LIN {X 0,Y 206.175,Z 893.981,A -85,B 0,C 180,E1 -23802.983,E2 -23802.983} C_VEL
LIN {X 0,Y 205.634,Z 894.543,A -85,B 0,C 180,E1 -23804.133,E2 -23804.133} C_VEL
LIN {X 0,Y 204.142,Z 895.622,A -85,B 0,C 180,E1 -23805.109,E2 -23805.109} C_VEL
LIN {X 0,Y 198.321,Z 899.43,A -85,B 0,C 180,E1 -23807.677,E2 -23807.677} C_VEL
LIN {X 0,Y 191.857,Z 903.186,A -85,B 0,C 180,E1 -23810.13,E2 -23810.13} C_VEL
LIN {X 0,Y 180.969,Z 908.434,A -85,B 0,C 180,E1 -23814.371,E2 -23814.371} C_VEL
LIN {X 0,Y 173.411,Z 911.413,A -85,B 0,C 180,E1 -23818.206,E2 -23818.206} C_VEL
LIN {X 0,Y 167.081,Z 913.319,A -85,B 0,C 180,E1 -23822.439,E2 -23822.439} C_VEL
LIN {X 0,Y 162.116,Z 914.142,A -85,B 0,C 180,E1 -23827.035,E2 -23827.035} C_VEL
LIN {X 0,Y 158.497,Z 913.842,A -85,B 0,C 180,E1 -23831.917,E2 -23831.917} C_VEL
LIN {X 0,Y 156.515,Z 912.431,A -85,B 0,C 180,E1 -23837.026,E2 -23837.026} C_VEL
LIN {X 0,Y 156.028,Z 909.791,A -85,B 0,C 180,E1 -23842.301,E2 -23842.301} C_VEL
LIN {X 0,Y 156.626,Z 905.821,A -85,B 0,C 180,E1 -23847.428,E2 -23847.428} C_VEL
LIN {X 0,Y 157.151,Z 904.017,A -85,B 0,C 180,E1 -23849.359,E2 -23849.359} C_VEL
LIN {X 0,Y 156.522,Z 907.281,A -85,B 0,C 180,E1 -23852.574,E2 -23852.574} C_VEL
LIN {X 0,Y 155.932,Z 911.226,A -85,B 0,C 180,E1 -23857.771,E2 -23857.771} C_VEL
LIN {X 0,Y 156.49,Z 913.74,A -85,B 0,C 180,E1 -23862.977,E2 -23862.977} C_VEL
LIN {X 0,Y 158.478,Z 915.084,A -85,B 0,C 180,E1 -23868.085,E2 -23868.085} C_VEL
LIN {X 0,Y 162.105,Z 915.337,A -85,B 0,C 180,E1 -23872.966,E2 -23872.966} C_VEL
LIN {X 0,Y 167.061,Z 914.483,A -85,B 0,C 180,E1 -23877.565,E2 -23877.565} C_VEL
LIN {X 0,Y 173.716,Z 912.427,A -85,B 0,C 180,E1 -23882.007,E2 -23882.007} C_VEL
LIN {X 0,Y 180.79,Z 909.587,A -85,B 0,C 180,E1 -23885.67,E2 -23885.67} C_VEL
LIN {X 0,Y 189.558,Z 905.487,A -85,B 0,C 180,E1 -23889.072,E2 -23889.072} C_VEL
LIN {X 0,Y 191.177,Z 904.654,A -85,B 0,C 180,E1 -23889.633,E2 -23889.633} C_VEL
LIN {X 0,Y 192.985,Z 903.559,A -85,B 0,C 180,E1 -23890.605,E2 -23890.605} C_VEL
LIN {X 0,Y 193.846,Z 902.733,A -85,B 0,C 180,E1 -23891.725,E2 -23891.725} C_VEL
LIN {X 0,Y 195.209,Z 900.797,A -85,B 0,C 180,E1 -23895.095,E2 -23895.095} C_VEL
LIN {X 0,Y 195.881,Z 900.333,A -85,B 0,C 180,E1 -23895.652,E2 -23895.652} C_VEL
LIN {X 0,Y 196.934,Z 899.471,A -85,B 0,C 180,E1 -23897.306,E2 -23897.306} C_VEL
LIN {X 0,Y 197.063,Z 899.174,A -85,B 0,C 180,E1 -23898.499,E2 -23898.499} C_VEL
LIN {X 0,Y 195.662,Z 899.564,A -85,B 0,C 180,E1 -23899.716,E2 -23899.716} C_VEL
LIN {X 0,Y 185.93,Z 902.848,A -85,B 0,C 180,E1 -23902.784,E2 -23902.784} C_VEL
LIN {X 0,Y 177.174,Z 904.928,A -85,B 0,C 180,E1 -23906.263,E2 -23906.263} C_VEL
LIN {X 0,Y 169.371,Z 905.875,A -85,B 0,C 180,E1 -23910.134,E2 -23910.134} C_VEL
LIN {X 0,Y 162.669,Z 905.677,A -85,B 0,C 180,E1 -23914.4,E2 -23914.4} C_VEL
LIN {X 0,Y 157.172,Z 904.299,A -85,B 0,C 180,E1 -23919.037,E2 -23919.037} C_VEL
LIN {X 0,Y 153.143,Z 901.751,A -85,B 0,C 180,E1 -23924.014,E2 -23924.014} C_VEL
LIN {X 0,Y 149.972,Z 897.499,A -85,B 0,C 180,E1 -23929.771,E2 -23929.771} C_VEL
LIN {X 0,Y 148.887,Z 892.858,A -85,B 0,C 180,E1 -23934.58,E2 -23934.58} C_VEL
LIN {X 0,Y 148.452,Z 887.997,A -85,B 0,C 180,E1 -23938.641,E2 -23938.641} C_VEL
LIN {X 0,Y 148.396,Z 882.089,A -85,B 0,C 180,E1 -23942.712,E2 -23942.712} C_VEL
LIN {X 0,Y 148.841,Z 873.681,A -85,B 0,C 180,E1 -23947.436,E2 -23947.436} C_VEL
LIN {X 0,Y 149.913,Z 863.17,A -85,B 0,C 180,E1 -23952.176,E2 -23952.176} C_VEL
LIN {X 0,Y 151.219,Z 853.005,A -85,B 0,C 180,E1 -23955.843,E2 -23955.843} C_VEL
LIN {X 0,Y 152.813,Z 841.876,A -85,B 0,C 180,E1 -23959.125,E2 -23959.125} C_VEL
LIN {X 0,Y 154.364,Z 831.542,A -85,B 0,C 180,E1 -23961.643,E2 -23961.643} C_VEL
LIN {X 0,Y 153.48,Z 825.601,A -85,B 0,C 180,E1 -23962.901,E2 -23962.901} C_VEL
LIN {X 0,Y 150.949,Z 811.534,A -85,B 0,C 180,E1 -23965.447,E2 -23965.447} C_VEL
LIN {X 0,Y 149.36,Z 802.881,A -85,B 0,C 180,E1 -23966.789,E2 -23966.789} C_VEL
LIN {X 0,Y 149.696,Z 802.832,A -85,B 0,C 180,E1 -23972.32,E2 -23972.32} C_VEL
LIN {X 0,Y 150.026,Z 802.795,A -85,B 0,C 180,E1 -23977.512,E2 -23977.512} C_VEL
LIN {X 0,Y 150.112,Z 802.781,A -85,B 0,C 180,E1 -23981.488,E2 -23981.488} C_VEL
LIN {X 0,Y 150.121,Z 802.784,A -85,B 0,C 180,E1 -23985.393,E2 -23985.393} C_VEL
LIN {X 0,Y 150.135,Z 802.777,A -85,B 0,C 180,E1 -23989.053,E2 -23989.053} C_VEL
LIN {X 0,Y 150.176,Z 802.777,A -85,B 0,C 180,E1 -23992.704,E2 -23992.704} C_VEL
LIN {X 0,Y 150.199,Z 802.77,A -85,B 0,C 180,E1 -23997.372,E2 -23997.372} C_VEL
LIN {X 0,Y 150.231,Z 802.771,A -85,B 0,C 180,E1 -24002.721,E2 -24002.721} C_VEL
LIN {X 0,Y 150.332,Z 802.755,A -85,B 0,C 180,E1 -24009.219,E2 -24009.219} C_VEL
LIN {X 0,Y 150.322,Z 802.759,A -85,B 0,C 180,E1 -24013.709,E2 -24013.709} C_VEL
LIN {X 0,Y 150.6,Z 802.723,A -85,B 0,C 180,E1 -24019.242,E2 -24019.242} C_VEL
LIN {X 0,Y 150.689,Z 802.714,A -85,B 0,C 180,E1 -24021.957,E2 -24021.957} C_VEL
LIN {X 0,Y 151.187,Z 802.654,A -85,B 0,C 180,E1 -24030,E2 -24030} C_VEL
LIN {X 0,Y 150.688,Z 802.714,A -85,B 0,C 180,E1 -24038.043,E2 -24038.043} C_VEL
LIN {X 0,Y 150.566,Z 802.727,A -85,B 0,C 180,E1 -24041.431,E2 -24041.431} C_VEL
LIN {X 0,Y 150.321,Z 802.759,A -85,B 0,C 180,E1 -24046.291,E2 -24046.291} C_VEL
LIN {X 0,Y 150.332,Z 802.755,A -85,B 0,C 180,E1 -24050.781,E2 -24050.781} C_VEL
LIN {X 0,Y 150.231,Z 802.771,A -85,B 0,C 180,E1 -24057.279,E2 -24057.279} C_VEL
LIN {X 0,Y 150.199,Z 802.77,A -85,B 0,C 180,E1 -24062.628,E2 -24062.628} C_VEL
LIN {X 0,Y 150.171,Z 802.777,A -85,B 0,C 180,E1 -24067.474,E2 -24067.474} C_VEL
LIN {X 0,Y 150.131,Z 802.78,A -85,B 0,C 180,E1 -24071.501,E2 -24071.501} C_VEL
LIN {X 0,Y 150.121,Z 802.786,A -85,B 0,C 180,E1 -24075.398,E2 -24075.398} C_VEL
LIN {X 0,Y 150.115,Z 802.781,A -85,B 0,C 180,E1 -24079.051,E2 -24079.051} C_VEL
LIN {X 0,Y 150.071,Z 802.79,A -85,B 0,C 180,E1 -24082.762,E2 -24082.762} C_VEL
LIN {X 0,Y 149.745,Z 802.826,A -85,B 0,C 180,E1 -24087.65,E2 -24087.65} C_VEL
LIN {X 0,Y 149.352,Z 802.883,A -85,B 0,C 180,E1 -24093.744,E2 -24093.744} C_VEL
LIN {X 0,Y 152.014,Z 817.45,A -85,B 0,C 180,E1 -24096.055,E2 -24096.055} C_VEL
LIN {X 0,Y 154.184,Z 829.238,A -85,B 0,C 180,E1 -24098.359,E2 -24098.359} C_VEL
LIN {X 0,Y 153.922,Z 833.391,A -85,B 0,C 180,E1 -24099.279,E2 -24099.279} C_VEL
LIN {X 0,Y 152.059,Z 845.938,A -85,B 0,C 180,E1 -24102.52,E2 -24102.52} C_VEL
LIN {X 0,Y 150.354,Z 858.144,A -85,B 0,C 180,E1 -24106.487,E2 -24106.487} C_VEL
LIN {X 0,Y 149.249,Z 868.043,A -85,B 0,C 180,E1 -24110.517,E2 -24110.517} C_VEL
LIN {X 0,Y 148.552,Z 876.986,A -85,B 0,C 180,E1 -24114.974,E2 -24114.974} C_VEL
LIN {X 0,Y 148.378,Z 883.073,A -85,B 0,C 180,E1 -24118.646,E2 -24118.646} C_VEL
LIN {X 0,Y 148.552,Z 888.659,A -85,B 0,C 180,E1 -24122.714,E2 -24122.714} C_VEL
LIN {X 0,Y 149.045,Z 893.275,A -85,B 0,C 180,E1 -24126.773,E2 -24126.773} C_VEL
LIN {X 0,Y 150.698,Z 898.09,A -85,B 0,C 180,E1 -24132.117,E2 -24132.117} C_VEL
LIN {X 0,Y 152.999,Z 900.836,A -85,B 0,C 180,E1 -24136.001,E2 -24136.001} C_VEL
LIN {X 0,Y 157.026,Z 903.417,A -85,B 0,C 180,E1 -24140.983,E2 -24140.983} C_VEL
LIN {X 0,Y 162.377,Z 904.818,A -85,B 0,C 180,E1 -24145.649,E2 -24145.649} C_VEL
LIN {X 0,Y 169.143,Z 905.029,A -85,B 0,C 180,E1 -24149.91,E2 -24149.91} C_VEL
LIN {X 0,Y 176.938,Z 904.069,A -85,B 0,C 180,E1 -24153.788,E2 -24153.788} C_VEL
LIN {X 0,Y 185.698,Z 901.963,A -85,B 0,C 180,E1 -24157.27,E2 -24157.27} C_VEL
LIN {X 0,Y 195.419,Z 898.667,A -85,B 0,C 180,E1 -24160.344,E2 -24160.344} C_VEL
LIN {X 0,Y 199.621,Z 897.048,A -85,B 0,C 180,E1 -24161.987,E2 -24161.987} C_VEL
LIN {X 0,Y 199.165,Z 897.595,A -85,B 0,C 180,E1 -24163.665,E2 -24163.665} C_VEL
LIN {X 0,Y 195.304,Z 899.854,A -85,B 0,C 180,E1 -24165.436,E2 -24165.436} C_VEL
LIN {X 0,Y 188.843,Z 903.25,A -85,B 0,C 180,E1 -24167.941,E2 -24167.941} C_VEL
LIN {X 0,Y 179.655,Z 907.311,A -85,B 0,C 180,E1 -24171.251,E2 -24171.251} C_VEL
LIN {X 0,Y 171.192,Z 910.365,A -85,B 0,C 180,E1 -24174.918,E2 -24174.918} C_VEL
LIN {X 0,Y 163.925,Z 912.373,A -85,B 0,C 180,E1 -24179.037,E2 -24179.037} C_VEL
LIN {X 0,Y 158.081,Z 913.344,A -85,B 0,C 180,E1 -24183.603,E2 -24183.603} C_VEL
LIN {X 0,Y 153.577,Z 913.247,A -85,B 0,C 180,E1 -24188.525,E2 -24188.525} C_VEL
LIN {X 0,Y 150.576,Z 912.07,A -85,B 0,C 180,E1 -24193.737,E2 -24193.737} C_VEL
LIN {X 0,Y 149.222,Z 909.786,A -85,B 0,C 180,E1 -24199.141,E2 -24199.141} C_VEL
LIN {X 0,Y 149.324,Z 906.261,A -85,B 0,C 180,E1 -24204.599,E2 -24204.599} C_VEL
LIN {X 0,Y 150.365,Z 901.963,A -85,B 0,C 180,E1 -24209.414,E2 -24209.414} C_VEL
LIN {X 0,Y 149.685,Z 905.392,A -85,B 0,C 180,E1 -24212.691,E2 -24212.691} C_VEL
LIN {X 0,Y 149.092,Z 909.56,A -85,B 0,C 180,E1 -24218.13,E2 -24218.13} C_VEL
LIN {X 0,Y 149.665,Z 912.382,A -85,B 0,C 180,E1 -24223.579,E2 -24223.579} C_VEL
LIN {X 0,Y 151.805,Z 914.025,A -85,B 0,C 180,E1 -24228.91,E2 -24228.91} C_VEL
LIN {X 0,Y 155.624,Z 914.615,A -85,B 0,C 180,E1 -24233.982,E2 -24233.982} C_VEL
LIN {X 0,Y 160.793,Z 914.136,A -85,B 0,C 180,E1 -24238.737,E2 -24238.737} C_VEL
LIN {X 0,Y 167.383,Z 912.62,A -85,B 0,C 180,E1 -24243.082,E2 -24243.082} C_VEL
LIN {X 0,Y 175.094,Z 910.094,A -85,B 0,C 180,E1 -24247.019,E2 -24247.019} C_VEL
LIN {X 0,Y 186.539,Z 905.456,A -85,B 0,C 180,E1 -24251.249,E2 -24251.249} C_VEL
LIN {X 0,Y 191.223,Z 903.172,A -85,B 0,C 180,E1 -24252.838,E2 -24252.838} C_VEL
LIN {X 0,Y 193.164,Z 902.101,A -85,B 0,C 180,E1 -24253.732,E2 -24253.732} C_VEL
LIN {X 0,Y 195.881,Z 900.333,A -85,B 0,C 180,E1 -24255.652,E2 -24255.652} C_VEL
LIN {X 0,Y 196.105,Z 900.056,A -85,B 0,C 180,E1 -24256.328,E2 -24256.328} C_VEL
LIN {X 0,Y 195.068,Z 900.298,A -85,B 0,C 180,E1 -24257.177,E2 -24257.177} C_VEL
LIN {X 0,Y 192.271,Z 901.204,A -85,B 0,C 180,E1 -24258.224,E2 -24258.224} C_VEL
LIN {X 0,Y 182.927,Z 903.94,A -85,B 0,C 180,E1 -24260.65,E2 -24260.65} C_VEL
LIN {X 0,Y 174.086,Z 905.806,A -85,B 0,C 180,E1 -24263.845,E2 -24263.845} C_VEL
LIN {X 0,Y 167.253,Z 906.544,A -85,B 0,C 180,E1 -24266.886,E2 -24266.886} C_VEL
LIN {X 0,Y 159.638,Z 906.493,A -85,B 0,C 180,E1 -24271.033,E2 -24271.033} C_VEL
LIN {X 0,Y 153.32,Z 905.309,A -85,B 0,C 180,E1 -24275.632,E2 -24275.632} C_VEL
LIN {X 0,Y 148.3,Z 902.979,A -85,B 0,C 180,E1 -24280.623,E2 -24280.623} C_VEL
LIN {X 0,Y 144.557,Z 899.455,A -85,B 0,C 180,E1 -24285.928,E2 -24285.928} C_VEL
LIN {X 0,Y 142.436,Z 894.647,A -85,B 0,C 180,E1 -24291.485,E2 -24291.485} C_VEL
LIN {X 0,Y 141.713,Z 890.153,A -85,B 0,C 180,E1 -24295.731,E2 -24295.731} C_VEL
LIN {X 0,Y 141.429,Z 883.627,A -85,B 0,C 180,E1 -24300.709,E2 -24300.709} C_VEL
LIN {X 0,Y 141.609,Z 875.558,A -85,B 0,C 180,E1 -24305.694,E2 -24305.694} C_VEL
LIN {X 0,Y 142.321,Z 867.055,A -85,B 0,C 180,E1 -24309.95,E2 -24309.95} C_VEL
LIN {X 0,Y 143.54,Z 856.768,A -85,B 0,C 180,E1 -24314.168,E2 -24314.168} C_VEL
LIN {X 0,Y 145.201,Z 845.463,A -85,B 0,C 180,E1 -24317.97,E2 -24317.97} C_VEL
LIN {X 0,Y 147.081,Z 832.613,A -85,B 0,C 180,E1 -24321.364,E2 -24321.364} C_VEL
LIN {X 0,Y 147.267,Z 831.185,A -85,B 0,C 180,E1 -24321.703,E2 -24321.703} C_VEL
LIN {X 0,Y 144.927,Z 818.339,A -85,B 0,C 180,E1 -24324.364,E2 -24324.364} C_VEL
LIN {X 0,Y 142.461,Z 804.577,A -85,B 0,C 180,E1 -24326.702,E2 -24326.702} C_VEL
LIN {X 0,Y 142.316,Z 803.759,A -85,B 0,C 180,E1 -24326.823,E2 -24326.823} C_VEL
LIN {X 0,Y 142.693,Z 803.707,A -85,B 0,C 180,E1 -24333.144,E2 -24333.144} C_VEL
LIN {X 0,Y 142.957,Z 803.677,A -85,B 0,C 180,E1 -24338.132,E2 -24338.132} C_VEL
LIN {X 0,Y 143.024,Z 803.668,A -85,B 0,C 180,E1 -24343.463,E2 -24343.463} C_VEL
LIN {X 0,Y 143.034,Z 803.664,A -85,B 0,C 180,E1 -24347.474,E2 -24347.474} C_VEL
LIN {X 0,Y 143.073,Z 803.661,A -85,B 0,C 180,E1 -24351.803,E2 -24351.803} C_VEL
LIN {X 0,Y 143.167,Z 803.646,A -85,B 0,C 180,E1 -24357.317,E2 -24357.317} C_VEL
LIN {X 0,Y 143.175,Z 803.649,A -85,B 0,C 180,E1 -24362.068,E2 -24362.068} C_VEL
LIN {X 0,Y 143.259,Z 803.634,A -85,B 0,C 180,E1 -24368.755,E2 -24368.755} C_VEL
LIN {X 0,Y 143.261,Z 803.639,A -85,B 0,C 180,E1 -24372.882,E2 -24372.882} C_VEL
LIN {X 0,Y 143.526,Z 803.604,A -85,B 0,C 180,E1 -24378.705,E2 -24378.705} C_VEL
LIN {X 0,Y 143.612,Z 803.597,A -85,B 0,C 180,E1 -24381.558,E2 -24381.558} C_VEL
LIN {X 0,Y 144.145,Z 803.531,A -85,B 0,C 180,E1 -24390,E2 -24390} C_VEL
LIN {X 0,Y 143.611,Z 803.597,A -85,B 0,C 180,E1 -24398.442,E2 -24398.442} C_VEL
LIN {X 0,Y 143.492,Z 803.608,A -85,B 0,C 180,E1 -24401.62,E2 -24401.62} C_VEL
LIN {X 0,Y 143.26,Z 803.639,A -85,B 0,C 180,E1 -24407.118,E2 -24407.118} C_VEL
LIN {X 0,Y 143.259,Z 803.634,A -85,B 0,C 180,E1 -24411.245,E2 -24411.245} C_VEL
LIN {X 0,Y 143.175,Z 803.649,A -85,B 0,C 180,E1 -24417.932,E2 -24417.932} C_VEL
LIN {X 0,Y 143.151,Z 803.652,A -85,B 0,C 180,E1 -24423.43,E2 -24423.43} C_VEL
LIN {X 0,Y 143.051,Z 803.659,A -85,B 0,C 180,E1 -24429.694,E2 -24429.694} C_VEL
LIN {X 0,Y 143.029,Z 803.669,A -85,B 0,C 180,E1 -24433.466,E2 -24433.466} C_VEL
LIN {X 0,Y 143.025,Z 803.666,A -85,B 0,C 180,E1 -24437.483,E2 -24437.483} C_VEL
LIN {X 0,Y 142.993,Z 803.672,A -85,B 0,C 180,E1 -24441.85,E2 -24441.85} C_VEL
LIN {X 0,Y 142.726,Z 803.703,A -85,B 0,C 180,E1 -24447.207,E2 -24447.207} C_VEL
LIN {X 0,Y 142.306,Z 803.76,A -85,B 0,C 180,E1 -24453.707,E2 -24453.707} C_VEL
LIN {X 0,Y 144.854,Z 817.542,A -85,B 0,C 180,E1 -24456.007,E2 -24456.007} C_VEL
LIN {X 0,Y 147.172,Z 830.38,A -85,B 0,C 180,E1 -24458.65,E2 -24458.65} C_VEL
LIN {X 0,Y 145.418,Z 842.37,A -85,B 0,C 180,E1 -24461.694,E2 -24461.694} C_VEL
LIN {X 0,Y 143.858,Z 853.197,A -85,B 0,C 180,E1 -24465.142,E2 -24465.142} C_VEL
LIN {X 0,Y 142.738,Z 862.359,A -85,B 0,C 180,E1 -24468.644,E2 -24468.644} C_VEL
LIN {X 0,Y 141.843,Z 871.49,A -85,B 0,C 180,E1 -24472.836,E2 -24472.836} C_VEL
LIN {X 0,Y 141.448,Z 879.161,A -85,B 0,C 180,E1 -24477.155,E2 -24477.155} C_VEL
LIN {X 0,Y 141.482,Z 885.478,A -85,B 0,C 180,E1 -24481.426,E2 -24481.426} C_VEL
LIN {X 0,Y 142.023,Z 891.791,A -85,B 0,C 180,E1 -24486.721,E2 -24486.721} C_VEL
LIN {X 0,Y 143.213,Z 896.221,A -85,B 0,C 180,E1 -24491.323,E2 -24491.323} C_VEL
LIN {X 0,Y 146.208,Z 900.417,A -85,B 0,C 180,E1 -24496.766,E2 -24496.766} C_VEL
LIN {X 0,Y 150.422,Z 903.381,A -85,B 0,C 180,E1 -24501.951,E2 -24501.951} C_VEL
LIN {X 0,Y 156.029,Z 905.169,A -85,B 0,C 180,E1 -24506.774,E2 -24506.774} C_VEL
LIN {X 0,Y 163.075,Z 905.786,A -85,B 0,C 180,E1 -24511.145,E2 -24511.145} C_VEL
LIN {X 0,Y 171.171,Z 905.283,A -85,B 0,C 180,E1 -24515.089,E2 -24515.089} C_VEL
LIN {X 0,Y 180.248,Z 903.671,A -85,B 0,C 180,E1 -24518.601,E2 -24518.601} C_VEL
LIN {X 0,Y 190.279,Z 900.899,A -85,B 0,C 180,E1 -24521.672,E2 -24521.672} C_VEL
LIN {X 0,Y 192.457,Z 900.35,A -85,B 0,C 180,E1 -24523.084,E2 -24523.084} C_VEL
LIN {X 0,Y 186.032,Z 903.406,A -85,B 0,C 180,E1 -24525.661,E2 -24525.661} C_VEL
LIN {X 0,Y 178.944,Z 906.271,A -85,B 0,C 180,E1 -24528.112,E2 -24528.112} C_VEL
LIN {X 0,Y 169.673,Z 909.366,A -85,B 0,C 180,E1 -24531.588,E2 -24531.588} C_VEL
LIN {X 0,Y 161.542,Z 911.45,A -85,B 0,C 180,E1 -24535.558,E2 -24535.558} C_VEL
LIN {X 0,Y 154.641,Z 912.53,A -85,B 0,C 180,E1 -24540.005,E2 -24540.005} C_VEL
LIN {X 0,Y 149.204,Z 912.593,A -85,B 0,C 180,E1 -24544.917,E2 -24544.917} C_VEL
LIN {X 0,Y 145.204,Z 911.608,A -85,B 0,C 180,E1 -24550.196,E2 -24550.196} C_VEL
LIN {X 0,Y 142.964,Z 909.582,A -85,B 0,C 180,E1 -24555.771,E2 -24555.771} C_VEL
LIN {X 0,Y 142.367,Z 905.815,A -85,B 0,C 180,E1 -24562.359,E2 -24562.359} C_VEL
LIN {X 0,Y 143.021,Z 901.853,A -85,B 0,C 180,E1 -24567.183,E2 -24567.183} C_VEL
LIN {X 0,Y 143.623,Z 899.76,A -85,B 0,C 180,E1 -24569.387,E2 -24569.387} C_VEL
LIN {X 0,Y 142.899,Z 903.323,A -85,B 0,C 180,E1 -24572.819,E2 -24572.819} C_VEL
LIN {X 0,Y 142.258,Z 908.003,A -85,B 0,C 180,E1 -24578.845,E2 -24578.845} C_VEL
LIN {X 0,Y 142.889,Z 910.883,A -85,B 0,C 180,E1 -24584.237,E2 -24584.237} C_VEL
LIN {X 0,Y 145.189,Z 912.859,A -85,B 0,C 180,E1 -24589.806,E2 -24589.806} C_VEL
LIN {X 0,Y 149.195,Z 913.779,A -85,B 0,C 180,E1 -24595.085,E2 -24595.085} C_VEL
LIN {X 0,Y 154.617,Z 913.665,A -85,B 0,C 180,E1 -24600,E2 -24600} C_VEL
LIN {X 0,Y 161.481,Z 912.552,A -85,B 0,C 180,E1 -24604.457,E2 -24604.457} C_VEL
LIN {X 0,Y 169.487,Z 910.453,A -85,B 0,C 180,E1 -24608.462,E2 -24608.462} C_VEL
LIN {X 0,Y 178.841,Z 907.349,A -85,B 0,C 180,E1 -24611.917,E2 -24611.917} C_VEL
LIN {X 0,Y 183.762,Z 905.432,A -85,B 0,C 180,E1 -24613.505,E2 -24613.505} C_VEL
LIN {X 0,Y 187.934,Z 903.513,A -85,B 0,C 180,E1 -24615.278,E2 -24615.278} C_VEL
LIN {X 0,Y 190.382,Z 902.031,A -85,B 0,C 180,E1 -24617.587,E2 -24617.587} C_VEL
LIN {X 0,Y 190.27,Z 901.919,A -85,B 0,C 180,E1 -24618.326,E2 -24618.326} C_VEL
LIN {X 0,Y 182.927,Z 903.94,A -85,B 0,C 180,E1 -24620.65,E2 -24620.65} C_VEL
LIN {X 0,Y 178.486,Z 905.059,A -85,B 0,C 180,E1 -24621.846,E2 -24621.846} C_VEL
LIN {X 0,Y 170.216,Z 906.554,A -85,B 0,C 180,E1 -24623.577,E2 -24623.577} C_VEL
LIN {X 0,Y 162.198,Z 907.34,A -85,B 0,C 180,E1 -24625.531,E2 -24625.531} C_VEL
LIN {X 0,Y 158.238,Z 907.324,A -85,B 0,C 180,E1 -24627.079,E2 -24627.079} C_VEL
LIN {X 0,Y 150.025,Z 906.252,A -85,B 0,C 180,E1 -24632.063,E2 -24632.063} C_VEL
LIN {X 0,Y 144.036,Z 904.094,A -85,B 0,C 180,E1 -24637.021,E2 -24637.021} C_VEL
LIN {X 0,Y 139.605,Z 900.811,A -85,B 0,C 180,E1 -24642.416,E2 -24642.416} C_VEL
LIN {X 0,Y 136.365,Z 896.323,A -85,B 0,C 180,E1 -24648.1,E2 -24648.1} C_VEL
LIN {X 0,Y 134.975,Z 890.46,A -85,B 0,C 180,E1 -24654.019,E2 -24654.019} C_VEL
LIN {X 0,Y 134.517,Z 884.032,A -85,B 0,C 180,E1 -24659.249,E2 -24659.249} C_VEL
LIN {X 0,Y 134.615,Z 876.025,A -85,B 0,C 180,E1 -24664.476,E2 -24664.476} C_VEL
LIN {X 0,Y 135.186,Z 867.676,A -85,B 0,C 180,E1 -24668.97,E2 -24668.97} C_VEL
LIN {X 0,Y 136.084,Z 859.354,A -85,B 0,C 180,E1 -24672.676,E2 -24672.676} C_VEL
LIN {X 0,Y 137.758,Z 847.338,A -85,B 0,C 180,E1 -24677.055,E2 -24677.055} C_VEL
LIN {X 0,Y 139.595,Z 835.13,A -85,B 0,C 180,E1 -24680.632,E2 -24680.632} C_VEL
LIN {X 0,Y 140.085,Z 830.844,A -85,B 0,C 180,E1 -24681.712,E2 -24681.712} C_VEL
LIN {X 0,Y 137.632,Z 817.679,A -85,B 0,C 180,E1 -24684.532,E2 -24684.532} C_VEL
LIN {X 0,Y 135.289,Z 804.634,A -85,B 0,C 180,E1 -24686.823,E2 -24686.823} C_VEL
LIN {X 0,Y 135.669,Z 804.583,A -85,B 0,C 180,E1 -24694.02,E2 -24694.02} C_VEL
LIN {X 0,Y 135.946,Z 804.545,A -85,B 0,C 180,E1 -24699.154,E2 -24699.154} C_VEL
LIN {X 0,Y 135.969,Z 804.547,A -85,B 0,C 180,E1 -24703.644,E2 -24703.644} C_VEL
LIN {X 0,Y 135.979,Z 804.543,A -85,B 0,C 180,E1 -24707.786,E2 -24707.786} C_VEL
LIN {X 0,Y 136.022,Z 804.539,A -85,B 0,C 180,E1 -24711.682,E2 -24711.682} C_VEL
LIN {X 0,Y 136.076,Z 804.532,A -85,B 0,C 180,E1 -24715.721,E2 -24715.721} C_VEL
LIN {X 0,Y 136.132,Z 804.527,A -85,B 0,C 180,E1 -24722.313,E2 -24722.313} C_VEL
LIN {X 0,Y 136.226,Z 804.511,A -85,B 0,C 180,E1 -24728.83,E2 -24728.83} C_VEL
LIN {X 0,Y 136.227,Z 804.513,A -85,B 0,C 180,E1 -24735.051,E2 -24735.051} C_VEL
LIN {X 0,Y 136.418,Z 804.49,A -85,B 0,C 180,E1 -24738.177,E2 -24738.177} C_VEL
LIN {X 0,Y 136.538,Z 804.477,A -85,B 0,C 180,E1 -24741.117,E2 -24741.117} C_VEL
LIN {X 0,Y 137.102,Z 804.408,A -85,B 0,C 180,E1 -24750,E2 -24750} C_VEL
LIN {X 0,Y 136.537,Z 804.477,A -85,B 0,C 180,E1 -24758.883,E2 -24758.883} C_VEL
LIN {X 0,Y 136.407,Z 804.491,A -85,B 0,C 180,E1 -24761.893,E2 -24761.893} C_VEL
LIN {X 0,Y 136.18,Z 804.521,A -85,B 0,C 180,E1 -24768.038,E2 -24768.038} C_VEL
LIN {X 0,Y 136.182,Z 804.516,A -85,B 0,C 180,E1 -24771.74,E2 -24771.74} C_VEL
LIN {X 0,Y 136.085,Z 804.533,A -85,B 0,C 180,E1 -24778.611,E2 -24778.611} C_VEL
LIN {X 0,Y 136.063,Z 804.535,A -85,B 0,C 180,E1 -24784.624,E2 -24784.624} C_VEL
LIN {X 0,Y 136.024,Z 804.536,A -85,B 0,C 180,E1 -24789.199,E2 -24789.199} C_VEL
LIN {X 0,Y 135.973,Z 804.547,A -85,B 0,C 180,E1 -24793.651,E2 -24793.651} C_VEL
LIN {X 0,Y 135.968,Z 804.544,A -85,B 0,C 180,E1 -24797.787,E2 -24797.787} C_VEL
LIN {X 0,Y 135.944,Z 804.549,A -85,B 0,C 180,E1 -24801.661,E2 -24801.661} C_VEL
LIN {X 0,Y 135.739,Z 804.574,A -85,B 0,C 180,E1 -24805.936,E2 -24805.936} C_VEL
LIN {X 0,Y 135.262,Z 804.637,A -85,B 0,C 180,E1 -24813.743,E2 -24813.743} C_VEL
LIN {X 0,Y 137.711,Z 817.957,A -85,B 0,C 180,E1 -24816.08,E2 -24816.08} C_VEL
LIN {X 0,Y 139.965,Z 829.977,A -85,B 0,C 180,E1 -24818.655,E2 -24818.655} C_VEL
LIN {X 0,Y 138.298,Z 842.003,A -85,B 0,C 180,E1 -24821.868,E2 -24821.868} C_VEL
LIN {X 0,Y 136.597,Z 853.921,A -85,B 0,C 180,E1 -24825.857,E2 -24825.857} C_VEL
LIN {X 0,Y 135.493,Z 863.316,A -85,B 0,C 180,E1 -24829.694,E2 -24829.694} C_VEL
LIN {X 0,Y 134.744,Z 872.033,A -85,B 0,C 180,E1 -24834.015,E2 -24834.015} C_VEL
LIN {X 0,Y 134.473,Z 879.583,A -85,B 0,C 180,E1 -24838.506,E2 -24838.506} C_VEL
LIN {X 0,Y 134.626,Z 885.808,A -85,B 0,C 180,E1 -24842.995,E2 -24842.995} C_VEL
LIN {X 0,Y 135.158,Z 891,A -85,B 0,C 180,E1 -24847.472,E2 -24847.472} C_VEL
LIN {X 0,Y 136.949,Z 896.511,A -85,B 0,C 180,E1 -24853.355,E2 -24853.355} C_VEL
LIN {X 0,Y 139.459,Z 899.853,A -85,B 0,C 180,E1 -24857.603,E2 -24857.603} C_VEL
LIN {X 0,Y 143.877,Z 903.158,A -85,B 0,C 180,E1 -24863.006,E2 -24863.006} C_VEL
LIN {X 0,Y 149.735,Z 905.335,A -85,B 0,C 180,E1 -24867.996,E2 -24867.996} C_VEL
LIN {X 0,Y 157.073,Z 906.397,A -85,B 0,C 180,E1 -24872.477,E2 -24872.477} C_VEL
LIN {X 0,Y 165.486,Z 906.347,A -85,B 0,C 180,E1 -24876.484,E2 -24876.484} C_VEL
LIN {X 0,Y 174.878,Z 905.206,A -85,B 0,C 180,E1 -24880.019,E2 -24880.019} C_VEL
LIN {X 0,Y 179.927,Z 904.233,A -85,B 0,C 180,E1 -24881.61,E2 -24881.61} C_VEL
LIN {X 0,Y 183.378,Z 903.563,A -85,B 0,C 180,E1 -24883.266,E2 -24883.266} C_VEL
LIN {X 0,Y 178.683,Z 905.342,A -85,B 0,C 180,E1 -24884.929,E2 -24884.929} C_VEL
LIN {X 0,Y 168.853,Z 908.417,A -85,B 0,C 180,E1 -24888.244,E2 -24888.244} C_VEL
LIN {X 0,Y 159.794,Z 910.548,A -85,B 0,C 180,E1 -24891.994,E2 -24891.994} C_VEL
LIN {X 0,Y 150.963,Z 911.785,A -85,B 0,C 180,E1 -24896.932,E2 -24896.932} C_VEL
LIN {X 0,Y 145.522,Z 911.899,A -85,B 0,C 180,E1 -24901.121,E2 -24901.121} C_VEL
LIN {X 0,Y 140.553,Z 911.093,A -85,B 0,C 180,E1 -24906.42,E2 -24906.42} C_VEL
LIN {X 0,Y 137.211,Z 909.263,A -85,B 0,C 180,E1 -24912.102,E2 -24912.102} C_VEL
LIN {X 0,Y 135.671,Z 906.365,A -85,B 0,C 180,E1 -24918.041,E2 -24918.041} C_VEL
LIN {X 0,Y 135.766,Z 902.244,A -85,B 0,C 180,E1 -24924.057,E2 -24924.057} C_VEL
LIN {X 0,Y 136.951,Z 897.368,A -85,B 0,C 180,E1 -24929.357,E2 -24929.357} C_VEL
LIN {X 0,Y 136.162,Z 901.109,A -85,B 0,C 180,E1 -24932.959,E2 -24932.959} C_VEL
LIN {X 0,Y 135.494,Z 905.904,A -85,B 0,C 180,E1 -24938.952,E2 -24938.952} C_VEL
LIN {X 0,Y 136.158,Z 909.289,A -85,B 0,C 180,E1 -24944.956,E2 -24944.956} C_VEL
LIN {X 0,Y 138.617,Z 911.552,A -85,B 0,C 180,E1 -24950.788,E2 -24950.788} C_VEL
LIN {X 0,Y 142.84,Z 912.808,A -85,B 0,C 180,E1 -24956.284,E2 -24956.284} C_VEL
LIN {X 0,Y 148.523,Z 913.056,A -85,B 0,C 180,E1 -24961.367,E2 -24961.367} C_VEL
LIN {X 0,Y 155.685,Z 912.337,A -85,B 0,C 180,E1 -24965.934,E2 -24965.934} C_VEL
LIN {X 0,Y 164.005,Z 910.672,A -85,B 0,C 180,E1 -24970,E2 -24970} C_VEL
LIN {X 0,Y 173.648,Z 908.04,A -85,B 0,C 180,E1 -24973.475,E2 -24973.475} C_VEL
LIN {X 0,Y 178.711,Z 906.372,A -85,B 0,C 180,E1 -24975.062,E2 -24975.062} C_VEL
LIN {X 0,Y 182.552,Z 904.787,A -85,B 0,C 180,E1 -24977.01,E2 -24977.01} C_VEL
LIN {X 0,Y 180.183,Z 905.148,A -85,B 0,C 180,E1 -24978.462,E2 -24978.462} C_VEL
LIN {X 0,Y 170.274,Z 906.827,A -85,B 0,C 180,E1 -24981.745,E2 -24981.745} C_VEL
LIN {X 0,Y 161.402,Z 907.4,A -85,B 0,C 180,E1 -24985.521,E2 -24985.521} C_VEL
LIN {X 0,Y 158.238,Z 907.324,A -85,B 0,C 180,E1 -24987.079,E2 -24987.079} C_VEL
LIN {X 0,Y 154.39,Z 907.156,A -85,B 0,C 180,E1 -24988.727,E2 -24988.727} C_VEL
LIN {X 0,Y 147.03,Z 906.374,A -85,B 0,C 180,E1 -24991.246,E2 -24991.246} C_VEL
LIN {X 0,Y 140.219,Z 904.867,A -85,B 0,C 180,E1 -24994.035,E2 -24994.035} C_VEL
LIN {X 0,Y 137.326,Z 903.61,A -85,B 0,C 180,E1 -24996.083,E2 -24996.083} C_VEL
LIN {X 0,Y 131.849,Z 899.004,A -85,B 0,C 180,E1 -25002.949,E2 -25002.949} C_VEL
LIN {X 0,Y 129.057,Z 893.968,A -85,B 0,C 180,E1 -25008.809,E2 -25008.809} C_VEL
LIN {X 0,Y 128.053,Z 889.023,A -85,B 0,C 180,E1 -25013.695,E2 -25013.695} C_VEL
LIN {X 0,Y 127.587,Z 882.217,A -85,B 0,C 180,E1 -25019.208,E2 -25019.208} C_VEL
LIN {X 0,Y 127.66,Z 875.117,A -85,B 0,C 180,E1 -25023.943,E2 -25023.943} C_VEL
LIN {X 0,Y 128.188,Z 866.905,A -85,B 0,C 180,E1 -25028.471,E2 -25028.471} C_VEL
LIN {X 0,Y 129.117,Z 858.06,A -85,B 0,C 180,E1 -25032.572,E2 -25032.572} C_VEL
LIN {X 0,Y 130.633,Z 847.009,A -85,B 0,C 180,E1 -25036.805,E2 -25036.805} C_VEL
LIN {X 0,Y 132.508,Z 834.637,A -85,B 0,C 180,E1 -25040.568,E2 -25040.568} C_VEL
LIN {X 0,Y 132.896,Z 831.853,A -85,B 0,C 180,E1 -25041.316,E2 -25041.316} C_VEL
LIN {X 0,Y 132.176,Z 826.883,A -85,B 0,C 180,E1 -25042.522,E2 -25042.522} C_VEL
LIN {X 0,Y 129.762,Z 813.906,A -85,B 0,C 180,E1 -25045.265,E2 -25045.265} C_VEL
LIN {X 0,Y 128.262,Z 805.509,A -85,B 0,C 180,E1 -25046.818,E2 -25046.818} C_VEL
LIN {X 0,Y 128.654,Z 805.459,A -85,B 0,C 180,E1 -25054.974,E2 -25054.974} C_VEL
LIN {X 0,Y 128.891,Z 805.423,A -85,B 0,C 180,E1 -25060.863,E2 -25060.863} C_VEL
LIN {X 0,Y 128.906,Z 805.428,A -85,B 0,C 180,E1 -25065.13,E2 -25065.13} C_VEL
LIN {X 0,Y 128.931,Z 805.417,A -85,B 0,C 180,E1 -25069.736,E2 -25069.736} C_VEL
LIN {X 0,Y 128.974,Z 805.42,A -85,B 0,C 180,E1 -25074.817,E2 -25074.817} C_VEL
LIN {X 0,Y 129.01,Z 805.411,A -85,B 0,C 180,E1 -25080.64,E2 -25080.64} C_VEL
LIN {X 0,Y 129.099,Z 805.397,A -85,B 0,C 180,E1 -25087.6,E2 -25087.6} C_VEL
LIN {X 0,Y 129.151,Z 805.394,A -85,B 0,C 180,E1 -25094.212,E2 -25094.212} C_VEL
LIN {X 0,Y 129.337,Z 805.37,A -85,B 0,C 180,E1 -25097.967,E2 -25097.967} C_VEL
LIN {X 0,Y 129.461,Z 805.358,A -85,B 0,C 180,E1 -25100.627,E2 -25100.627} C_VEL
LIN {X 0,Y 130.057,Z 805.286,A -85,B 0,C 180,E1 -25110,E2 -25110} C_VEL
LIN {X 0,Y 129.461,Z 805.358,A -85,B 0,C 180,E1 -25119.373,E2 -25119.373} C_VEL
LIN {X 0,Y 129.291,Z 805.373,A -85,B 0,C 180,E1 -25122.558,E2 -25122.558} C_VEL
LIN {X 0,Y 129.106,Z 805.402,A -85,B 0,C 180,E1 -25129.064,E2 -25129.064} C_VEL
LIN {X 0,Y 129.099,Z 805.397,A -85,B 0,C 180,E1 -25132.4,E2 -25132.4} C_VEL
LIN {X 0,Y 129.01,Z 805.411,A -85,B 0,C 180,E1 -25139.36,E2 -25139.36} C_VEL
LIN {X 0,Y 128.974,Z 805.42,A -85,B 0,C 180,E1 -25145.183,E2 -25145.183} C_VEL
LIN {X 0,Y 128.919,Z 805.419,A -85,B 0,C 180,E1 -25150.858,E2 -25150.858} C_VEL
LIN {X 0,Y 128.906,Z 805.429,A -85,B 0,C 180,E1 -25155.135,E2 -25155.135} C_VEL
LIN {X 0,Y 128.903,Z 805.422,A -85,B 0,C 180,E1 -25159.757,E2 -25159.757} C_VEL
LIN {X 0,Y 128.717,Z 805.451,A -85,B 0,C 180,E1 -25164.985,E2 -25164.985} C_VEL
LIN {X 0,Y 128.234,Z 805.511,A -85,B 0,C 180,E1 -25173.171,E2 -25173.171} C_VEL
LIN {X 0,Y 128.23,Z 805.512,A -85,B 0,C 180,E1 -25173.792,E2 -25173.792} C_VEL
LIN {X 0,Y 130.86,Z 819.638,A -85,B 0,C 180,E1 -25176.475,E2 -25176.475} C_VEL
LIN {X 0,Y 132.708,Z 829.312,A -85,B 0,C 180,E1 -25178.652,E2 -25178.652} C_VEL
LIN {X 0,Y 132.551,Z 832.429,A -85,B 0,C 180,E1 -25179.439,E2 -25179.439} C_VEL
LIN {X 0,Y 130.684,Z 845.092,A -85,B 0,C 180,E1 -25183.202,E2 -25183.202} C_VEL
LIN {X 0,Y 129.225,Z 856.437,A -85,B 0,C 180,E1 -25187.439,E2 -25187.439} C_VEL
LIN {X 0,Y 128.031,Z 868.076,A -85,B 0,C 180,E1 -25192.861,E2 -25192.861} C_VEL
LIN {X 0,Y 127.59,Z 876.312,A -85,B 0,C 180,E1 -25197.636,E2 -25197.636} C_VEL
LIN {X 0,Y 127.706,Z 884.102,A -85,B 0,C 180,E1 -25203.158,E2 -25203.158} C_VEL
LIN {X 0,Y 128.279,Z 889.565,A -85,B 0,C 180,E1 -25207.876,E2 -25207.876} C_VEL
LIN {X 0,Y 130.131,Z 895.495,A -85,B 0,C 180,E1 -25214.069,E2 -25214.069} C_VEL
LIN {X 0,Y 133.769,Z 900.113,A -85,B 0,C 180,E1 -25219.971,E2 -25219.971} C_VEL
LIN {X 0,Y 137.393,Z 902.763,A -85,B 0,C 180,E1 -25224.159,E2 -25224.159} C_VEL
LIN {X 0,Y 143.524,Z 905.35,A -85,B 0,C 180,E1 -25229.322,E2 -25229.322} C_VEL
LIN {X 0,Y 151.142,Z 906.843,A -85,B 0,C 180,E1 -25233.92,E2 -25233.92} C_VEL
LIN {X 0,Y 159.882,Z 907.25,A -85,B 0,C 180,E1 -25237.984,E2 -25237.984} C_VEL
LIN {X 0,Y 169.591,Z 906.592,A -85,B 0,C 180,E1 -25241.536,E2 -25241.536} C_VEL
LIN {X 0,Y 173.766,Z 906.109,A -85,B 0,C 180,E1 -25243.28,E2 -25243.28} C_VEL
LIN {X 0,Y 163.648,Z 908.711,A -85,B 0,C 180,E1 -25246.596,E2 -25246.596} C_VEL
LIN {X 0,Y 154.28,Z 910.396,A -85,B 0,C 180,E1 -25250.376,E2 -25250.376} C_VEL
LIN {X 0,Y 144.728,Z 911.151,A -85,B 0,C 180,E1 -25255.646,E2 -25255.646} C_VEL
LIN {X 0,Y 139.388,Z 910.943,A -85,B 0,C 180,E1 -25259.721,E2 -25259.721} C_VEL
LIN {X 0,Y 134.18,Z 909.796,A -85,B 0,C 180,E1 -25265.227,E2 -25265.227} C_VEL
LIN {X 0,Y 130.629,Z 907.655,A -85,B 0,C 180,E1 -25271.167,E2 -25271.167} C_VEL
LIN {X 0,Y 128.978,Z 904.468,A -85,B 0,C 180,E1 -25277.411,E2 -25277.411} C_VEL
LIN {X 0,Y 129.068,Z 900.031,A -85,B 0,C 180,E1 -25283.748,E2 -25283.748} C_VEL
LIN {X 0,Y 130.313,Z 894.915,A -85,B 0,C 180,E1 -25289.421,E2 -25289.421} C_VEL
LIN {X 0,Y 129.181,Z 900.202,A -85,B 0,C 180,E1 -25294.681,E2 -25294.681} C_VEL
LIN {X 0,Y 128.797,Z 904.725,A -85,B 0,C 180,E1 -25300.812,E2 -25300.812} C_VEL
LIN {X 0,Y 129.527,Z 907.501,A -85,B 0,C 180,E1 -25305.741,E2 -25305.741} C_VEL
LIN {X 0,Y 132.136,Z 910.09,A -85,B 0,C 180,E1 -25311.859,E2 -25311.859} C_VEL
LIN {X 0,Y 136.571,Z 911.662,A -85,B 0,C 180,E1 -25317.59,E2 -25317.59} C_VEL
LIN {X 0,Y 142.527,Z 912.278,A -85,B 0,C 180,E1 -25322.848,E2 -25322.848} C_VEL
LIN {X 0,Y 149.997,Z 911.963,A -85,B 0,C 180,E1 -25327.525,E2 -25327.525} C_VEL
LIN {X 0,Y 158.633,Z 910.71,A -85,B 0,C 180,E1 -25331.648,E2 -25331.648} C_VEL
LIN {X 0,Y 168.578,Z 908.548,A -85,B 0,C 180,E1 -25335.132,E2 -25335.132} C_VEL
LIN {X 0,Y 173.697,Z 907.127,A -85,B 0,C 180,E1 -25336.745,E2 -25336.745} C_VEL
LIN {X 0,Y 169.798,Z 907.53,A -85,B 0,C 180,E1 -25338.526,E2 -25338.526} C_VEL
LIN {X 0,Y 160.121,Z 908.174,A -85,B 0,C 180,E1 -25342.083,E2 -25342.083} C_VEL
LIN {X 0,Y 151.375,Z 907.776,A -85,B 0,C 180,E1 -25346.139,E2 -25346.139} C_VEL
LIN {X 0,Y 143.798,Z 906.301,A -85,B 0,C 180,E1 -25350.739,E2 -25350.739} C_VEL
LIN {X 0,Y 137.326,Z 903.61,A -85,B 0,C 180,E1 -25356.083,E2 -25356.083} C_VEL
LIN {X 0,Y 134.663,Z 902.212,A -85,B 0,C 180,E1 -25358.209,E2 -25358.209} C_VEL
LIN {X 0,Y 129.102,Z 899.269,A -85,B 0,C 180,E1 -25361.53,E2 -25361.53} C_VEL
LIN {X 0,Y 124.119,Z 895.623,A -85,B 0,C 180,E1 -25365.069,E2 -25365.069} C_VEL
LIN {X 0,Y 122.461,Z 893.246,A -85,B 0,C 180,E1 -25367.484,E2 -25367.484} C_VEL
LIN {X 0,Y 121.175,Z 887.37,A -85,B 0,C 180,E1 -25373.335,E2 -25373.335} C_VEL
LIN {X 0,Y 120.696,Z 880.189,A -85,B 0,C 180,E1 -25379.163,E2 -25379.163} C_VEL
LIN {X 0,Y 120.845,Z 871.315,A -85,B 0,C 180,E1 -25385.001,E2 -25385.001} C_VEL
LIN {X 0,Y 121.602,Z 862.013,A -85,B 0,C 180,E1 -25389.981,E2 -25389.981} C_VEL
LIN {X 0,Y 122.938,Z 850.691,A -85,B 0,C 180,E1 -25394.904,E2 -25394.904} C_VEL
LIN {X 0,Y 124.566,Z 839.258,A -85,B 0,C 180,E1 -25398.926,E2 -25398.926} C_VEL
LIN {X 0,Y 125.804,Z 831.274,A -85,B 0,C 180,E1 -25401.288,E2 -25401.288} C_VEL
LIN {X 0,Y 123.411,Z 818.436,A -85,B 0,C 180,E1 -25404.333,E2 -25404.333} C_VEL
LIN {X 0,Y 121.215,Z 806.387,A -85,B 0,C 180,E1 -25406.791,E2 -25406.791} C_VEL
LIN {X 0,Y 121.629,Z 806.334,A -85,B 0,C 180,E1 -25415.293,E2 -25415.293} C_VEL
LIN {X 0,Y 121.821,Z 806.305,A -85,B 0,C 180,E1 -25421.411,E2 -25421.411} C_VEL
LIN {X 0,Y 121.859,Z 806.3,A -85,B 0,C 180,E1 -25428.563,E2 -25428.563} C_VEL
LIN {X 0,Y 121.926,Z 806.298,A -85,B 0,C 180,E1 -25434.801,E2 -25434.801} C_VEL
LIN {X 0,Y 121.922,Z 806.294,A -85,B 0,C 180,E1 -25439.836,E2 -25439.836} C_VEL
LIN {X 0,Y 121.973,Z 806.286,A -85,B 0,C 180,E1 -25446.213,E2 -25446.213} C_VEL
LIN {X 0,Y 122.013,Z 806.285,A -85,B 0,C 180,E1 -25449.781,E2 -25449.781} C_VEL
LIN {X 0,Y 122.182,Z 806.257,A -85,B 0,C 180,E1 -25456.698,E2 -25456.698} C_VEL
LIN {X 0,Y 122.388,Z 806.24,A -85,B 0,C 180,E1 -25460.08,E2 -25460.08} C_VEL
LIN {X 0,Y 122.551,Z 806.215,A -85,B 0,C 180,E1 -25466.712,E2 -25466.712} C_VEL
LIN {X 0,Y 123.011,Z 806.163,A -85,B 0,C 180,E1 -25470,E2 -25470} C_VEL
LIN {X 0,Y 122.398,Z 806.237,A -85,B 0,C 180,E1 -25476.594,E2 -25476.594} C_VEL
LIN {X 0,Y 122.388,Z 806.24,A -85,B 0,C 180,E1 -25479.92,E2 -25479.92} C_VEL
LIN {X 0,Y 122.182,Z 806.257,A -85,B 0,C 180,E1 -25483.302,E2 -25483.302} C_VEL
LIN {X 0,Y 122.013,Z 806.285,A -85,B 0,C 180,E1 -25490.219,E2 -25490.219} C_VEL
LIN {X 0,Y 121.973,Z 806.286,A -85,B 0,C 180,E1 -25493.787,E2 -25493.787} C_VEL
LIN {X 0,Y 121.922,Z 806.294,A -85,B 0,C 180,E1 -25500.164,E2 -25500.164} C_VEL
LIN {X 0,Y 121.891,Z 806.301,A -85,B 0,C 180,E1 -25506.182,E2 -25506.182} C_VEL
LIN {X 0,Y 121.859,Z 806.3,A -85,B 0,C 180,E1 -25511.437,E2 -25511.437} C_VEL
LIN {X 0,Y 121.827,Z 806.304,A -85,B 0,C 180,E1 -25518.586,E2 -25518.586} C_VEL
LIN {X 0,Y 121.685,Z 806.327,A -85,B 0,C 180,E1 -25524.726,E2 -25524.726} C_VEL
LIN {X 0,Y 121.217,Z 806.385,A -85,B 0,C 180,E1 -25532.37,E2 -25532.37} C_VEL
LIN {X 0,Y 121.223,Z 806.544,A -85,B 0,C 180,E1 -25534.001,E2 -25534.001} C_VEL
LIN {X 0,Y 123.852,Z 820.421,A -85,B 0,C 180,E1 -25536.765,E2 -25536.765} C_VEL
LIN {X 0,Y 125.685,Z 830.288,A -85,B 0,C 180,E1 -25539.12,E2 -25539.12} C_VEL
LIN {X 0,Y 123.808,Z 843.319,A -85,B 0,C 180,E1 -25543.09,E2 -25543.09} C_VEL
LIN {X 0,Y 122.199,Z 855.737,A -85,B 0,C 180,E1 -25547.882,E2 -25547.882} C_VEL
LIN {X 0,Y 121.215,Z 865.292,A -85,B 0,C 180,E1 -25552.458,E2 -25552.458} C_VEL
LIN {X 0,Y 120.732,Z 873.966,A -85,B 0,C 180,E1 -25557.501,E2 -25557.501} C_VEL
LIN {X 0,Y 120.807,Z 881.15,A -85,B 0,C 180,E1 -25562.504,E2 -25562.504} C_VEL
LIN {X 0,Y 121.44,Z 887.966,A -85,B 0,C 180,E1 -25568.322,E2 -25568.322} C_VEL
LIN {X 0,Y 123.384,Z 894.265,A -85,B 0,C 180,E1 -25574.855,E2 -25574.855} C_VEL
LIN {X 0,Y 127.185,Z 899.28,A -85,B 0,C 180,E1 -25581.053,E2 -25581.053} C_VEL
LIN {X 0,Y 133.984,Z 903.829,A -85,B 0,C 180,E1 -25588.173,E2 -25588.173} C_VEL
LIN {X 0,Y 141.184,Z 906.281,A -85,B 0,C 180,E1 -25593.204,E2 -25593.204} C_VEL
LIN {X 0,Y 149.727,Z 907.67,A -85,B 0,C 180,E1 -25597.607,E2 -25597.607} C_VEL
LIN {X 0,Y 160.622,Z 907.986,A -85,B 0,C 180,E1 -25601.941,E2 -25601.941} C_VEL
LIN {X 0,Y 163.758,Z 907.857,A -85,B 0,C 180,E1 -25603.148,E2 -25603.148} C_VEL
LIN {X 0,Y 153.594,Z 909.553,A -85,B 0,C 180,E1 -25606.658,E2 -25606.658} C_VEL
LIN {X 0,Y 144.537,Z 910.339,A -85,B 0,C 180,E1 -25610.794,E2 -25610.794} C_VEL
LIN {X 0,Y 136.716,Z 910.203,A -85,B 0,C 180,E1 -25615.565,E2 -25615.565} C_VEL
LIN {X 0,Y 130.431,Z 909.169,A -85,B 0,C 180,E1 -25620.991,E2 -25620.991} C_VEL
LIN {X 0,Y 125.757,Z 907.193,A -85,B 0,C 180,E1 -25626.971,E2 -25626.971} C_VEL
LIN {X 0,Y 123.008,Z 904.246,A -85,B 0,C 180,E1 -25633.401,E2 -25633.401} C_VEL
LIN {X 0,Y 122.196,Z 900.187,A -85,B 0,C 180,E1 -25640.064,E2 -25640.064} C_VEL
LIN {X 0,Y 122.997,Z 894.738,A -85,B 0,C 180,E1 -25646.724,E2 -25646.724} C_VEL
LIN {X 0,Y 123.719,Z 892.259,A -85,B 0,C 180,E1 -25649.39,E2 -25649.39} C_VEL
LIN {X 0,Y 122.542,Z 897.753,A -85,B 0,C 180,E1 -25654.935,E2 -25654.935} C_VEL
LIN {X 0,Y 122.105,Z 901.615,A -85,B 0,C 180,E1 -25659.943,E2 -25659.943} C_VEL
LIN {X 0,Y 122.944,Z 905.557,A -85,B 0,C 180,E1 -25666.608,E2 -25666.608} C_VEL
LIN {X 0,Y 125.745,Z 908.442,A -85,B 0,C 180,E1 -25673.031,E2 -25673.031} C_VEL
LIN {X 0,Y 130.405,Z 910.353,A -85,B 0,C 180,E1 -25679.015,E2 -25679.015} C_VEL
LIN {X 0,Y 138.281,Z 911.398,A -85,B 0,C 180,E1 -25685.587,E2 -25685.587} C_VEL
LIN {X 0,Y 148.775,Z 911.1,A -85,B 0,C 180,E1 -25691.403,E2 -25691.403} C_VEL
LIN {X 0,Y 158.439,Z 909.833,A -85,B 0,C 180,E1 -25695.213,E2 -25695.213} C_VEL
LIN {X 0,Y 163.652,Z 908.861,A -85,B 0,C 180,E1 -25696.892,E2 -25696.892} C_VEL
LIN {X 0,Y 157.266,Z 908.961,A -85,B 0,C 180,E1 -25699.439,E2 -25699.439} C_VEL
LIN {X 0,Y 149.96,Z 908.631,A -85,B 0,C 180,E1 -25702.461,E2 -25702.461} C_VEL
LIN {X 0,Y 141.424,Z 907.264,A -85,B 0,C 180,E1 -25706.86,E2 -25706.86} C_VEL
LIN {X 0,Y 134.225,Z 904.839,A -85,B 0,C 180,E1 -25711.882,E2 -25711.882} C_VEL
LIN {X 0,Y 128.471,Z 901.352,A -85,B 0,C 180,E1 -25717.481,E2 -25717.481} C_VEL
LIN {X 0,Y 124.216,Z 896.718,A -85,B 0,C 180,E1 -25723.564,E2 -25723.564} C_VEL
LIN {X 0,Y 122.461,Z 893.246,A -85,B 0,C 180,E1 -25727.484,E2 -25727.484} C_VEL
LIN {X 0,Y 121.098,Z 890.735,A -85,B 0,C 180,E1 -25729.909,E2 -25729.909} C_VEL
LIN {X 0,Y 117.632,Z 885.829,A -85,B 0,C 180,E1 -25733.685,E2 -25733.685} C_VEL
LIN {X 0,Y 115.016,Z 881.439,A -85,B 0,C 180,E1 -25736.731,E2 -25736.731} C_VEL
LIN {X 0,Y 113.929,Z 877.986,A -85,B 0,C 180,E1 -25739.129,E2 -25739.129} C_VEL
LIN {X 0,Y 113.84,Z 876.834,A -85,B 0,C 180,E1 -25739.954,E2 -25739.954} C_VEL
LIN {X 0,Y 114.028,Z 868.577,A -85,B 0,C 180,E1 -25745.301,E2 -25745.301} C_VEL
LIN {X 0,Y 114.946,Z 858.097,A -85,B 0,C 180,E1 -25750.918,E2 -25750.918} C_VEL
LIN {X 0,Y 116.156,Z 847.908,A -85,B 0,C 180,E1 -25755.346,E2 -25755.346} C_VEL
LIN {X 0,Y 117.723,Z 837.184,A -85,B 0,C 180,E1 -25759.165,E2 -25759.165} C_VEL
LIN {X 0,Y 118.592,Z 831.775,A -85,B 0,C 180,E1 -25760.825,E2 -25760.825} C_VEL
LIN {X 0,Y 118.148,Z 828.128,A -85,B 0,C 180,E1 -25761.821,E2 -25761.821} C_VEL
LIN {X 0,Y 115.566,Z 815.036,A -85,B 0,C 180,E1 -25764.917,E2 -25764.917} C_VEL
LIN {X 0,Y 114.215,Z 807.259,A -85,B 0,C 180,E1 -25766.552,E2 -25766.552} C_VEL
LIN {X 0,Y 114.366,Z 807.236,A -85,B 0,C 180,E1 -25773.573,E2 -25773.573} C_VEL
LIN {X 0,Y 114.622,Z 807.206,A -85,B 0,C 180,E1 -25777.813,E2 -25777.813} C_VEL
LIN {X 0,Y 114.742,Z 807.189,A -85,B 0,C 180,E1 -25782.692,E2 -25782.692} C_VEL
LIN {X 0,Y 114.781,Z 807.183,A -85,B 0,C 180,E1 -25787.66,E2 -25787.66} C_VEL
LIN {X 0,Y 114.791,Z 807.185,A -85,B 0,C 180,E1 -25792.736,E2 -25792.736} C_VEL
LIN {X 0,Y 114.854,Z 807.17,A -85,B 0,C 180,E1 -25798.937,E2 -25798.937} C_VEL
LIN {X 0,Y 114.938,Z 807.162,A -85,B 0,C 180,E1 -25806.508,E2 -25806.508} C_VEL
LIN {X 0,Y 114.977,Z 807.162,A -85,B 0,C 180,E1 -25812.204,E2 -25812.204} C_VEL
LIN {X 0,Y 115.301,Z 807.121,A -85,B 0,C 180,E1 -25819.464,E2 -25819.464} C_VEL
LIN {X 0,Y 115.478,Z 807.095,A -85,B 0,C 180,E1 -25826.511,E2 -25826.511} C_VEL
LIN {X 0,Y 115.963,Z 807.041,A -85,B 0,C 180,E1 -25830,E2 -25830} C_VEL
LIN {X 0,Y 115.341,Z 807.116,A -85,B 0,C 180,E1 -25837,E2 -25837} C_VEL
LIN {X 0,Y 115.198,Z 807.128,A -85,B 0,C 180,E1 -25842.562,E2 -25842.562} C_VEL
LIN {X 0,Y 114.976,Z 807.162,A -85,B 0,C 180,E1 -25847.796,E2 -25847.796} C_VEL
LIN {X 0,Y 114.938,Z 807.162,A -85,B 0,C 180,E1 -25853.492,E2 -25853.492} C_VEL
LIN {X 0,Y 114.854,Z 807.17,A -85,B 0,C 180,E1 -25861.063,E2 -25861.063} C_VEL
LIN {X 0,Y 114.78,Z 807.185,A -85,B 0,C 180,E1 -25867.756,E2 -25867.756} C_VEL
LIN {X 0,Y 114.773,Z 807.185,A -85,B 0,C 180,E1 -25872.715,E2 -25872.715} C_VEL
LIN {X 0,Y 114.754,Z 807.186,A -85,B 0,C 180,E1 -25877.653,E2 -25877.653} C_VEL
LIN {X 0,Y 114.654,Z 807.202,A -85,B 0,C 180,E1 -25882.833,E2 -25882.833} C_VEL
LIN {X 0,Y 114.242,Z 807.247,A -85,B 0,C 180,E1 -25889.459,E2 -25889.459} C_VEL
LIN {X 0,Y 114.19,Z 807.26,A -85,B 0,C 180,E1 -25894.179,E2 -25894.179} C_VEL
LIN {X 0,Y 116.805,Z 820.978,A -85,B 0,C 180,E1 -25897.1,E2 -25897.1} C_VEL
LIN {X 0,Y 118.48,Z 829.255,A -85,B 0,C 180,E1 -25899.155,E2 -25899.155} C_VEL
LIN {X 0,Y 117.086,Z 840.164,A -85,B 0,C 180,E1 -25902.539,E2 -25902.539} C_VEL
LIN {X 0,Y 115.48,Z 852.101,A -85,B 0,C 180,E1 -25907.165,E2 -25907.165} C_VEL
LIN {X 0,Y 114.496,Z 861.659,A -85,B 0,C 180,E1 -25911.706,E2 -25911.706} C_VEL
LIN {X 0,Y 113.923,Z 871.443,A -85,B 0,C 180,E1 -25917.352,E2 -25917.352} C_VEL
LIN {X 0,Y 114.022,Z 880.102,A -85,B 0,C 180,E1 -25923.537,E2 -25923.537} C_VEL
LIN {X 0,Y 114.646,Z 886.192,A -85,B 0,C 180,E1 -25928.819,E2 -25928.819} C_VEL
LIN {X 0,Y 116.597,Z 892.715,A -85,B 0,C 180,E1 -25935.562,E2 -25935.562} C_VEL
LIN {X 0,Y 120.685,Z 898.219,A -85,B 0,C 180,E1 -25942.246,E2 -25942.246} C_VEL
LIN {X 0,Y 124.639,Z 901.46,A -85,B 0,C 180,E1 -25946.817,E2 -25946.817} C_VEL
LIN {X 0,Y 131.383,Z 904.843,A -85,B 0,C 180,E1 -25952.342,E2 -25952.342} C_VEL
LIN {X 0,Y 139.609,Z 907.177,A -85,B 0,C 180,E1 -25957.167,E2 -25957.167} C_VEL
LIN {X 0,Y 148.992,Z 908.49,A -85,B 0,C 180,E1 -25961.332,E2 -25961.332} C_VEL
LIN {X 0,Y 152.369,Z 908.678,A -85,B 0,C 180,E1 -25962.592,E2 -25962.592} C_VEL
LIN {X 0,Y 152.127,Z 908.88,A -85,B 0,C 180,E1 -25963.49,E2 -25963.49} C_VEL
LIN {X 0,Y 143.656,Z 909.516,A -85,B 0,C 180,E1 -25966.771,E2 -25966.771} C_VEL
LIN {X 0,Y 133.028,Z 909.278,A -85,B 0,C 180,E1 -25972.421,E2 -25972.421} C_VEL
LIN {X 0,Y 124.395,Z 907.695,A -85,B 0,C 180,E1 -25979.438,E2 -25979.438} C_VEL
LIN {X 0,Y 119.465,Z 905.391,A -85,B 0,C 180,E1 -25985.682,E2 -25985.682} C_VEL
LIN {X 0,Y 116.097,Z 901.176,A -85,B 0,C 180,E1 -25994.192,E2 -25994.192} C_VEL
LIN {X 0,Y 115.69,Z 896.503,A -85,B 0,C 180,E1 -26001.265,E2 -26001.265} C_VEL
LIN {X 0,Y 116.446,Z 892.031,A -85,B 0,C 180,E1 -26006.54,E2 -26006.54} C_VEL
LIN {X 0,Y 117.23,Z 889.38,A -85,B 0,C 180,E1 -26009.356,E2 -26009.356} C_VEL
LIN {X 0,Y 115.955,Z 895.171,A -85,B 0,C 180,E1 -26015.216,E2 -26015.216} C_VEL
LIN {X 0,Y 115.542,Z 899.975,A -85,B 0,C 180,E1 -26021.611,E2 -26021.611} C_VEL
LIN {X 0,Y 116.427,Z 903.495,A -85,B 0,C 180,E1 -26027.567,E2 -26027.567} C_VEL
LIN {X 0,Y 119.455,Z 906.658,A -85,B 0,C 180,E1 -26034.32,E2 -26034.32} C_VEL
LIN {X 0,Y 124.375,Z 908.862,A -85,B 0,C 180,E1 -26040.568,E2 -26040.568} C_VEL
LIN {X 0,Y 132.576,Z 910.338,A -85,B 0,C 180,E1 -26047.325,E2 -26047.325} C_VEL
LIN {X 0,Y 143.548,Z 910.544,A -85,B 0,C 180,E1 -26053.27,E2 -26053.27} C_VEL
LIN {X 0,Y 148.333,Z 910.237,A -85,B 0,C 180,E1 -26055.292,E2 -26055.292} C_VEL
LIN {X 0,Y 153.524,Z 909.719,A -85,B 0,C 180,E1 -26057.092,E2 -26057.092} C_VEL
LIN {X 0,Y 144.403,Z 908.95,A -85,B 0,C 180,E1 -26060.747,E2 -26060.747} C_VEL
LIN {X 0,Y 135.55,Z 907.145,A -85,B 0,C 180,E1 -26065.224,E2 -26065.224} C_VEL
LIN {X 0,Y 128.029,Z 904.331,A -85,B 0,C 180,E1 -26070.39,E2 -26070.39} C_VEL
LIN {X 0,Y 122.013,Z 900.474,A -85,B 0,C 180,E1 -26076.218,E2 -26076.218} C_VEL
LIN {X 0,Y 117.543,Z 895.427,A -85,B 0,C 180,E1 -26082.602,E2 -26082.602} C_VEL
LIN {X 0,Y 114.983,Z 889.171,A -85,B 0,C 180,E1 -26089.431,E2 -26089.431} C_VEL
LIN {X 0,Y 114.063,Z 882.459,A -85,B 0,C 180,E1 -26095.579,E2 -26095.579} C_VEL
LIN {X 0,Y 113.84,Z 876.834,A -85,B 0,C 180,E1 -26099.954,E2 -26099.954} C_VEL
LIN {X 0,Y 113.244,Z 873.234,A -85,B 0,C 180,E1 -26102.292,E2 -26102.292} C_VEL
LIN {X 0,Y 111.864,Z 869.294,A -85,B 0,C 180,E1 -26104.445,E2 -26104.445} C_VEL
LIN {X 0,Y 108.472,Z 859.378,A -85,B 0,C 180,E1 -26109.26,E2 -26109.26} C_VEL
LIN {X 0,Y 108.234,Z 854.918,A -85,B 0,C 180,E1 -26111.376,E2 -26111.376} C_VEL
LIN {X 0,Y 109.748,Z 843.024,A -85,B 0,C 180,E1 -26116.553,E2 -26116.553} C_VEL
LIN {X 0,Y 111.522,Z 830.764,A -85,B 0,C 180,E1 -26120.757,E2 -26120.757} C_VEL
LIN {X 0,Y 109.063,Z 818.238,A -85,B 0,C 180,E1 -26124.045,E2 -26124.045} C_VEL
LIN {X 0,Y 107.173,Z 808.136,A -85,B 0,C 180,E1 -26126.353,E2 -26126.353} C_VEL
LIN {X 0,Y 107.181,Z 808.125,A -85,B 0,C 180,E1 -26131.635,E2 -26131.635} C_VEL
LIN {X 0,Y 107.555,Z 808.084,A -85,B 0,C 180,E1 -26138.36,E2 -26138.36} C_VEL
LIN {X 0,Y 107.657,Z 808.074,A -85,B 0,C 180,E1 -26145.892,E2 -26145.892} C_VEL
LIN {X 0,Y 107.686,Z 808.069,A -85,B 0,C 180,E1 -26151.545,E2 -26151.545} C_VEL
LIN {X 0,Y 107.792,Z 808.049,A -85,B 0,C 180,E1 -26158.56,E2 -26158.56} C_VEL
LIN {X 0,Y 107.9,Z 808.037,A -85,B 0,C 180,E1 -26166.995,E2 -26166.995} C_VEL
LIN {X 0,Y 107.999,Z 808.028,A -85,B 0,C 180,E1 -26174.912,E2 -26174.912} C_VEL
LIN {X 0,Y 108.219,Z 808.002,A -85,B 0,C 180,E1 -26178.765,E2 -26178.765} C_VEL
LIN {X 0,Y 108.282,Z 807.995,A -85,B 0,C 180,E1 -26182.541,E2 -26182.541} C_VEL
LIN {X 0,Y 108.888,Z 807.922,A -85,B 0,C 180,E1 -26190,E2 -26190} C_VEL
LIN {X 0,Y 108.281,Z 807.995,A -85,B 0,C 180,E1 -26197.459,E2 -26197.459} C_VEL
LIN {X 0,Y 108.131,Z 808.007,A -85,B 0,C 180,E1 -26202.877,E2 -26202.877} C_VEL
LIN {X 0,Y 107.877,Z 808.046,A -85,B 0,C 180,E1 -26209.011,E2 -26209.011} C_VEL
LIN {X 0,Y 107.847,Z 808.046,A -85,B 0,C 180,E1 -26214.182,E2 -26214.182} C_VEL
LIN {X 0,Y 107.78,Z 808.051,A -85,B 0,C 180,E1 -26222.047,E2 -26222.047} C_VEL
LIN {X 0,Y 107.686,Z 808.069,A -85,B 0,C 180,E1 -26228.455,E2 -26228.455} C_VEL
LIN {X 0,Y 107.648,Z 808.075,A -85,B 0,C 180,E1 -26235.903,E2 -26235.903} C_VEL
LIN {X 0,Y 107.592,Z 808.08,A -85,B 0,C 180,E1 -26241.615,E2 -26241.615} C_VEL
LIN {X 0,Y 107.5,Z 808.094,A -85,B 0,C 180,E1 -26243.962,E2 -26243.962} C_VEL
LIN {X 0,Y 107.227,Z 808.119,A -85,B 0,C 180,E1 -26248.437,E2 -26248.437} C_VEL
LIN {X 0,Y 107.171,Z 808.134,A -85,B 0,C 180,E1 -26254.503,E2 -26254.503} C_VEL
LIN {X 0,Y 109.855,Z 821.905,A -85,B 0,C 180,E1 -26257.618,E2 -26257.618} C_VEL
LIN {X 0,Y 111.381,Z 829.779,A -85,B 0,C 180,E1 -26259.698,E2 -26259.698} C_VEL
LIN {X 0,Y 109.651,Z 842.365,A -85,B 0,C 180,E1 -26264.033,E2 -26264.033} C_VEL
LIN {X 0,Y 108.279,Z 853.488,A -85,B 0,C 180,E1 -26268.776,E2 -26268.776} C_VEL
LIN {X 0,Y 107.344,Z 864.024,A -85,B 0,C 180,E1 -26274.368,E2 -26274.368} C_VEL
LIN {X 0,Y 107.085,Z 872.76,A -85,B 0,C 180,E1 -26280.004,E2 -26280.004} C_VEL
LIN {X 0,Y 107.403,Z 880.028,A -85,B 0,C 180,E1 -26285.637,E2 -26285.637} C_VEL
LIN {X 0,Y 108.186,Z 886.034,A -85,B 0,C 180,E1 -26291.242,E2 -26291.242} C_VEL
LIN {X 0,Y 110.946,Z 892.777,A -85,B 0,C 180,E1 -26298.469,E2 -26298.469} C_VEL
LIN {X 0,Y 115.535,Z 898.239,A -85,B 0,C 180,E1 -26305.206,E2 -26305.206} C_VEL
LIN {X 0,Y 121.725,Z 902.53,A -85,B 0,C 180,E1 -26311.311,E2 -26311.311} C_VEL
LIN {X 0,Y 129.583,Z 905.778,A -85,B 0,C 180,E1 -26316.63,E2 -26316.63} C_VEL
LIN {X 0,Y 138.766,Z 908.03,A -85,B 0,C 180,E1 -26321.182,E2 -26321.182} C_VEL
LIN {X 0,Y 140.959,Z 908.373,A -85,B 0,C 180,E1 -26322.101,E2 -26322.101} C_VEL
LIN {X 0,Y 141.915,Z 908.722,A -85,B 0,C 180,E1 -26323.443,E2 -26323.443} C_VEL
LIN {X 0,Y 133.919,Z 908.625,A -85,B 0,C 180,E1 -26326.981,E2 -26326.981} C_VEL
LIN {X 0,Y 125.428,Z 907.727,A -85,B 0,C 180,E1 -26331.949,E2 -26331.949} C_VEL
LIN {X 0,Y 118.5,Z 906.015,A -85,B 0,C 180,E1 -26337.739,E2 -26337.739} C_VEL
LIN {X 0,Y 113.272,Z 903.4,A -85,B 0,C 180,E1 -26344.258,E2 -26344.258} C_VEL
LIN {X 0,Y 110.102,Z 899.841,A -85,B 0,C 180,E1 -26351.388,E2 -26351.388} C_VEL
LIN {X 0,Y 109.129,Z 895.228,A -85,B 0,C 180,E1 -26358.86,E2 -26358.86} C_VEL
LIN {X 0,Y 109.986,Z 889.174,A -85,B 0,C 180,E1 -26366.336,E2 -26366.336} C_VEL
LIN {X 0,Y 110.84,Z 886.322,A -85,B 0,C 180,E1 -26369.319,E2 -26369.319} C_VEL
LIN {X 0,Y 109.457,Z 892.412,A -85,B 0,C 180,E1 -26375.527,E2 -26375.527} C_VEL
LIN {X 0,Y 109.098,Z 898.057,A -85,B 0,C 180,E1 -26383.227,E2 -26383.227} C_VEL
LIN {X 0,Y 111.379,Z 903.087,A -85,B 0,C 180,E1 -26392.247,E2 -26392.247} C_VEL
LIN {X 0,Y 115.642,Z 906.072,A -85,B 0,C 180,E1 -26399.09,E2 -26399.09} C_VEL
LIN {X 0,Y 121.731,Z 908.141,A -85,B 0,C 180,E1 -26405.264,E2 -26405.264} C_VEL
LIN {X 0,Y 129.4,Z 909.358,A -85,B 0,C 180,E1 -26410.674,E2 -26410.674} C_VEL
LIN {X 0,Y 141.881,Z 909.725,A -85,B 0,C 180,E1 -26416.679,E2 -26416.679} C_VEL
LIN {X 0,Y 142.147,Z 909.541,A -85,B 0,C 180,E1 -26417.593,E2 -26417.593} C_VEL
LIN {X 0,Y 134.234,Z 908.05,A -85,B 0,C 180,E1 -26421.073,E2 -26421.073} C_VEL
LIN {X 0,Y 125.718,Z 905.326,A -85,B 0,C 180,E1 -26426.008,E2 -26426.008} C_VEL
LIN {X 0,Y 118.546,Z 901.6,A -85,B 0,C 180,E1 -26431.684,E2 -26431.684} C_VEL
LIN {X 0,Y 113.164,Z 896.83,A -85,B 0,C 180,E1 -26438.119,E2 -26438.119} C_VEL
LIN {X 0,Y 109.288,Z 890.783,A -85,B 0,C 180,E1 -26445.091,E2 -26445.091} C_VEL
LIN {X 0,Y 107.601,Z 883.46,A -85,B 0,C 180,E1 -26452.49,E2 -26452.49} C_VEL
LIN {X 0,Y 107.062,Z 875.154,A -85,B 0,C 180,E1 -26459.295,E2 -26459.295} C_VEL
LIN {X 0,Y 107.164,Z 867.169,A -85,B 0,C 180,E1 -26464.698,E2 -26464.698} C_VEL
LIN {X 0,Y 108.086,Z 856.229,A -85,B 0,C 180,E1 -26470.741,E2 -26470.741} C_VEL
LIN {X 0,Y 108.234,Z 854.918,A -85,B 0,C 180,E1 -26471.376,E2 -26471.376} C_VEL
LIN {X 0,Y 108.306,Z 850.416,A -85,B 0,C 180,E1 -26473.409,E2 -26473.409} C_VEL
LIN {X 0,Y 107.776,Z 845.672,A -85,B 0,C 180,E1 -26475.301,E2 -26475.301} C_VEL
LIN {X 0,Y 105.666,Z 835.762,A -85,B 0,C 180,E1 -26478.748,E2 -26478.748} C_VEL
LIN {X 0,Y 104.082,Z 828.877,A -85,B 0,C 180,E1 -26480.829,E2 -26480.829} C_VEL
LIN {X 0,Y 101.451,Z 816.063,A -85,B 0,C 180,E1 -26484.245,E2 -26484.245} C_VEL
LIN {X 0,Y 100.167,Z 809.008,A -85,B 0,C 180,E1 -26486.002,E2 -26486.002} C_VEL
LIN {X 0,Y 100.207,Z 809,A -85,B 0,C 180,E1 -26494.125,E2 -26494.125} C_VEL
LIN {X 0,Y 100.5,Z 808.959,A -85,B 0,C 180,E1 -26499.714,E2 -26499.714} C_VEL
LIN {X 0,Y 100.626,Z 808.95,A -85,B 0,C 180,E1 -26505.699,E2 -26505.699} C_VEL
LIN {X 0,Y 100.623,Z 808.945,A -85,B 0,C 180,E1 -26511.053,E2 -26511.053} C_VEL
LIN {X 0,Y 100.688,Z 808.938,A -85,B 0,C 180,E1 -26516.879,E2 -26516.879} C_VEL
LIN {X 0,Y 100.78,Z 808.928,A -85,B 0,C 180,E1 -26525.265,E2 -26525.265} C_VEL
LIN {X 0,Y 100.796,Z 808.926,A -85,B 0,C 180,E1 -26529.597,E2 -26529.597} C_VEL
LIN {X 0,Y 101.118,Z 808.884,A -85,B 0,C 180,E1 -26537.965,E2 -26537.965} C_VEL
LIN {X 0,Y 101.219,Z 808.876,A -85,B 0,C 180,E1 -26542.018,E2 -26542.018} C_VEL
LIN {X 0,Y 101.816,Z 808.803,A -85,B 0,C 180,E1 -26550,E2 -26550} C_VEL
LIN {X 0,Y 101.218,Z 808.876,A -85,B 0,C 180,E1 -26557.982,E2 -26557.982} C_VEL
LIN {X 0,Y 101.05,Z 808.889,A -85,B 0,C 180,E1 -26563.192,E2 -26563.192} C_VEL
LIN {X 0,Y 100.796,Z 808.926,A -85,B 0,C 180,E1 -26570.403,E2 -26570.403} C_VEL
LIN {X 0,Y 100.768,Z 808.931,A -85,B 0,C 180,E1 -26574.96,E2 -26574.96} C_VEL
LIN {X 0,Y 100.688,Z 808.938,A -85,B 0,C 180,E1 -26583.121,E2 -26583.121} C_VEL
LIN {X 0,Y 100.635,Z 808.942,A -85,B 0,C 180,E1 -26589.814,E2 -26589.814} C_VEL
LIN {X 0,Y 100.622,Z 808.951,A -85,B 0,C 180,E1 -26595.703,E2 -26595.703} C_VEL
LIN {X 0,Y 100.538,Z 808.956,A -85,B 0,C 180,E1 -26601.019,E2 -26601.019} C_VEL
LIN {X 0,Y 100.218,Z 808.995,A -85,B 0,C 180,E1 -26607.302,E2 -26607.302} C_VEL
LIN {X 0,Y 100.182,Z 809.004,A -85,B 0,C 180,E1 -26614.905,E2 -26614.905} C_VEL
LIN {X 0,Y 103.118,Z 823.668,A -85,B 0,C 180,E1 -26618.515,E2 -26618.515} C_VEL
LIN {X 0,Y 104.223,Z 829.936,A -85,B 0,C 180,E1 -26620.3,E2 -26620.3} C_VEL
LIN {X 0,Y 102.549,Z 842.015,A -85,B 0,C 180,E1 -26624.732,E2 -26624.732} C_VEL
LIN {X 0,Y 101.264,Z 853.477,A -85,B 0,C 180,E1 -26630.012,E2 -26630.012} C_VEL
LIN {X 0,Y 100.447,Z 863.935,A -85,B 0,C 180,E1 -26635.992,E2 -26635.992} C_VEL
LIN {X 0,Y 100.358,Z 871.299,A -85,B 0,C 180,E1 -26641.007,E2 -26641.007} C_VEL
LIN {X 0,Y 100.823,Z 878.714,A -85,B 0,C 180,E1 -26647.011,E2 -26647.011} C_VEL
LIN {X 0,Y 101.905,Z 885.335,A -85,B 0,C 180,E1 -26653.433,E2 -26653.433} C_VEL
LIN {X 0,Y 105.477,Z 892.614,A -85,B 0,C 180,E1 -26661.502,E2 -26661.502} C_VEL
LIN {X 0,Y 110.776,Z 898.131,A -85,B 0,C 180,E1 -26668.417,E2 -26668.417} C_VEL
LIN {X 0,Y 115.79,Z 901.526,A -85,B 0,C 180,E1 -26673.115,E2 -26673.115} C_VEL
LIN {X 0,Y 123.987,Z 905.187,A -85,B 0,C 180,E1 -26678.577,E2 -26678.577} C_VEL
LIN {X 0,Y 131.971,Z 907.517,A -85,B 0,C 180,E1 -26682.527,E2 -26682.527} C_VEL
LIN {X 0,Y 130.881,Z 907.611,A -85,B 0,C 180,E1 -26683.914,E2 -26683.914} C_VEL
LIN {X 0,Y 120.034,Z 906.203,A -85,B 0,C 180,E1 -26689.905,E2 -26689.905} C_VEL
LIN {X 0,Y 112.75,Z 904.173,A -85,B 0,C 180,E1 -26695.875,E2 -26695.875} C_VEL
LIN {X 0,Y 107.214,Z 901.268,A -85,B 0,C 180,E1 -26702.686,E2 -26702.686} C_VEL
LIN {X 0,Y 103.319,Z 896.239,A -85,B 0,C 180,E1 -26712.245,E2 -26712.245} C_VEL
LIN {X 0,Y 102.767,Z 891.042,A -85,B 0,C 180,E1 -26720.156,E2 -26720.156} C_VEL
LIN {X 0,Y 104.14,Z 884.292,A -85,B 0,C 180,E1 -26728.066,E2 -26728.066} C_VEL
LIN {X 0,Y 104.517,Z 883.147,A -85,B 0,C 180,E1 -26729.278,E2 -26729.278} C_VEL
LIN {X 0,Y 103.051,Z 889.445,A -85,B 0,C 180,E1 -26735.872,E2 -26735.872} C_VEL
LIN {X 0,Y 102.669,Z 895.283,A -85,B 0,C 180,E1 -26743.862,E2 -26743.862} C_VEL
LIN {X 0,Y 105.179,Z 900.807,A -85,B 0,C 180,E1 -26753.636,E2 -26753.636} C_VEL
LIN {X 0,Y 109.731,Z 904.102,A -85,B 0,C 180,E1 -26760.823,E2 -26760.823} C_VEL
LIN {X 0,Y 116.16,Z 906.459,A -85,B 0,C 180,E1 -26767.231,E2 -26767.231} C_VEL
LIN {X 0,Y 124.211,Z 908.008,A -85,B 0,C 180,E1 -26772.764,E2 -26772.764} C_VEL
LIN {X 0,Y 130.892,Z 908.667,A -85,B 0,C 180,E1 -26776.168,E2 -26776.168} C_VEL
LIN {X 0,Y 132.111,Z 908.571,A -85,B 0,C 180,E1 -26777.583,E2 -26777.583} C_VEL
LIN {X 0,Y 124.203,Z 906.266,A -85,B 0,C 180,E1 -26781.502,E2 -26781.502} C_VEL
LIN {X 0,Y 114.164,Z 901.592,A -85,B 0,C 180,E1 -26788.445,E2 -26788.445} C_VEL
LIN {X 0,Y 108.031,Z 896.707,A -85,B 0,C 180,E1 -26794.981,E2 -26794.981} C_VEL
LIN {X 0,Y 103.489,Z 890.635,A -85,B 0,C 180,E1 -26802.2,E2 -26802.2} C_VEL
LIN {X 0,Y 101.029,Z 882.236,A -85,B 0,C 180,E1 -26810.991,E2 -26810.991} C_VEL
LIN {X 0,Y 100.408,Z 875.366,A -85,B 0,C 180,E1 -26816.987,E2 -26816.987} C_VEL
LIN {X 0,Y 100.324,Z 867.077,A -85,B 0,C 180,E1 -26823.008,E2 -26823.008} C_VEL
LIN {X 0,Y 100.957,Z 857.193,A -85,B 0,C 180,E1 -26829.007,E2 -26829.007} C_VEL
LIN {X 0,Y 102.143,Z 846.266,A -85,B 0,C 180,E1 -26834.311,E2 -26834.311} C_VEL
LIN {X 0,Y 103.741,Z 834.914,A -85,B 0,C 180,E1 -26838.829,E2 -26838.829} C_VEL
LIN {X 0,Y 104.355,Z 830.961,A -85,B 0,C 180,E1 -26840.187,E2 -26840.187} C_VEL
LIN {X 0,Y 104.082,Z 828.877,A -85,B 0,C 180,E1 -26840.829,E2 -26840.829} C_VEL
LIN {X 0,Y 102.686,Z 825.513,A -85,B 0,C 180,E1 -26841.74,E2 -26841.74} C_VEL
LIN {X 0,Y 98.667,Z 820.458,A -85,B 0,C 180,E1 -26842.919,E2 -26842.919} C_VEL
LIN {X 0,Y 94.773,Z 815.304,A -85,B 0,C 180,E1 -26844.101,E2 -26844.101} C_VEL
LIN {X 0,Y 93.52,Z 811.788,A -85,B 0,C 180,E1 -26844.94,E2 -26844.94} C_VEL
LIN {X 0,Y 93.191,Z 809.877,A -85,B 0,C 180,E1 -26845.478,E2 -26845.478} C_VEL
LIN {X 0,Y 93.149,Z 809.879,A -85,B 0,C 180,E1 -26853.907,E2 -26853.907} C_VEL
LIN {X 0,Y 93.448,Z 809.837,A -85,B 0,C 180,E1 -26861.229,E2 -26861.229} C_VEL
LIN {X 0,Y 93.526,Z 809.827,A -85,B 0,C 180,E1 -26868.709,E2 -26868.709} C_VEL
LIN {X 0,Y 93.585,Z 809.826,A -85,B 0,C 180,E1 -26875.689,E2 -26875.689} C_VEL
LIN {X 0,Y 93.662,Z 809.817,A -85,B 0,C 180,E1 -26884.204,E2 -26884.204} C_VEL
LIN {X 0,Y 93.678,Z 809.808,A -85,B 0,C 180,E1 -26887.968,E2 -26887.968} C_VEL
LIN {X 0,Y 93.975,Z 809.769,A -85,B 0,C 180,E1 -26896.441,E2 -26896.441} C_VEL
LIN {X 0,Y 94.15,Z 809.758,A -85,B 0,C 180,E1 -26901.414,E2 -26901.414} C_VEL
LIN {X 0,Y 94.746,Z 809.684,A -85,B 0,C 180,E1 -26910,E2 -26910} C_VEL
LIN {X 0,Y 94.149,Z 809.758,A -85,B 0,C 180,E1 -26918.586,E2 -26918.586} C_VEL
LIN {X 0,Y 93.975,Z 809.769,A -85,B 0,C 180,E1 -26923.559,E2 -26923.559} C_VEL
LIN {X 0,Y 93.678,Z 809.808,A -85,B 0,C 180,E1 -26932.032,E2 -26932.032} C_VEL
LIN {X 0,Y 93.614,Z 809.825,A -85,B 0,C 180,E1 -26936.772,E2 -26936.772} C_VEL
LIN {X 0,Y 93.585,Z 809.826,A -85,B 0,C 180,E1 -26944.311,E2 -26944.311} C_VEL
LIN {X 0,Y 93.519,Z 809.832,A -85,B 0,C 180,E1 -26952.559,E2 -26952.559} C_VEL
LIN {X 0,Y 93.468,Z 809.835,A -85,B 0,C 180,E1 -26958.757,E2 -26958.757} C_VEL
LIN {X 0,Y 93.209,Z 809.872,A -85,B 0,C 180,E1 -26966.038,E2 -26966.038} C_VEL
LIN {X 0,Y 93.197,Z 809.873,A -85,B 0,C 180,E1 -26975.455,E2 -26975.455} C_VEL
LIN {X 0,Y 96.483,Z 825.641,A -85,B 0,C 180,E1 -26979.637,E2 -26979.637} C_VEL
LIN {X 0,Y 97.11,Z 829.77,A -85,B 0,C 180,E1 -26980.929,E2 -26980.929} C_VEL
LIN {X 0,Y 95.466,Z 841.848,A -85,B 0,C 180,E1 -26985.755,E2 -26985.755} C_VEL
LIN {X 0,Y 94.297,Z 853.321,A -85,B 0,C 180,E1 -26991.432,E2 -26991.432} C_VEL
LIN {X 0,Y 93.735,Z 862.135,A -85,B 0,C 180,E1 -26996.781,E2 -26996.781} C_VEL
LIN {X 0,Y 93.781,Z 871.028,A -85,B 0,C 180,E1 -27003.226,E2 -27003.226} C_VEL
LIN {X 0,Y 94.458,Z 878.39,A -85,B 0,C 180,E1 -27009.641,E2 -27009.641} C_VEL
LIN {X 0,Y 97.048,Z 887.32,A -85,B 0,C 180,E1 -27019.023,E2 -27019.023} C_VEL
LIN {X 0,Y 101.744,Z 893.853,A -85,B 0,C 180,E1 -27026.683,E2 -27026.683} C_VEL
LIN {X 0,Y 109.996,Z 900.319,A -85,B 0,C 180,E1 -27035.107,E2 -27035.107} C_VEL
LIN {X 0,Y 120.916,Z 905.235,A -85,B 0,C 180,E1 -27041.949,E2 -27041.949} C_VEL
LIN {X 0,Y 122.057,Z 905.645,A -85,B 0,C 180,E1 -27042.523,E2 -27042.523} C_VEL
LIN {X 0,Y 121.657,Z 905.775,A -85,B 0,C 180,E1 -27043.773,E2 -27043.773} C_VEL
LIN {X 0,Y 110.791,Z 903.391,A -85,B 0,C 180,E1 -27050.628,E2 -27050.628} C_VEL
LIN {X 0,Y 104,Z 900.632,A -85,B 0,C 180,E1 -27057.274,E2 -27057.274} C_VEL
LIN {X 0,Y 98.338,Z 895.86,A -85,B 0,C 180,E1 -27066.854,E2 -27066.854} C_VEL
LIN {X 0,Y 96.479,Z 890.955,A -85,B 0,C 180,E1 -27075.229,E2 -27075.229} C_VEL
LIN {X 0,Y 96.881,Z 884.714,A -85,B 0,C 180,E1 -27083.753,E2 -27083.753} C_VEL
LIN {X 0,Y 98.274,Z 879.732,A -85,B 0,C 180,E1 -27089.232,E2 -27089.232} C_VEL
LIN {X 0,Y 96.698,Z 886.338,A -85,B 0,C 180,E1 -27096.259,E2 -27096.259} C_VEL
LIN {X 0,Y 96.277,Z 891.056,A -85,B 0,C 180,E1 -27102.65,E2 -27102.65} C_VEL
LIN {X 0,Y 97.536,Z 896.161,A -85,B 0,C 180,E1 -27111.117,E2 -27111.117} C_VEL
LIN {X 0,Y 101.296,Z 900.223,A -85,B 0,C 180,E1 -27119.056,E2 -27119.056} C_VEL
LIN {X 0,Y 107.161,Z 903.356,A -85,B 0,C 180,E1 -27126.175,E2 -27126.175} C_VEL
LIN {X 0,Y 114.799,Z 905.616,A -85,B 0,C 180,E1 -27132.332,E2 -27132.332} C_VEL
LIN {X 0,Y 121.184,Z 906.798,A -85,B 0,C 180,E1 -27136.068,E2 -27136.068} C_VEL
LIN {X 0,Y 122.221,Z 906.74,A -85,B 0,C 180,E1 -27137.585,E2 -27137.585} C_VEL
LIN {X 0,Y 112.223,Z 902.62,A -85,B 0,C 180,E1 -27143.488,E2 -27143.488} C_VEL
LIN {X 0,Y 104.803,Z 897.844,A -85,B 0,C 180,E1 -27149.801,E2 -27149.801} C_VEL
LIN {X 0,Y 99.071,Z 891.837,A -85,B 0,C 180,E1 -27157.251,E2 -27157.251} C_VEL
LIN {X 0,Y 95.518,Z 884.935,A -85,B 0,C 180,E1 -27165.073,E2 -27165.073} C_VEL
LIN {X 0,Y 94.101,Z 877.479,A -85,B 0,C 180,E1 -27172.486,E2 -27172.486} C_VEL
LIN {X 0,Y 93.602,Z 869.839,A -85,B 0,C 180,E1 -27178.92,E2 -27178.92} C_VEL
LIN {X 0,Y 93.828,Z 860.487,A -85,B 0,C 180,E1 -27185.368,E2 -27185.368} C_VEL
LIN {X 0,Y 94.759,Z 849.218,A -85,B 0,C 180,E1 -27191.764,E2 -27191.764} C_VEL
LIN {X 0,Y 96.243,Z 837.739,A -85,B 0,C 180,E1 -27196.979,E2 -27196.979} C_VEL
LIN {X 0,Y 97.201,Z 829.773,A -85,B 0,C 180,E1 -27199.956,E2 -27199.956} C_VEL
LIN {X 0,Y 94.423,Z 816.56,A -85,B 0,C 180,E1 -27203.735,E2 -27203.735} C_VEL
LIN {X 0,Y 93.52,Z 811.788,A -85,B 0,C 180,E1 -27204.94,E2 -27204.94} C_VEL
LIN {X 0,Y 93.046,Z 810.57,A -85,B 0,C 180,E1 -27205.7,E2 -27205.7} C_VEL
LIN {X 0,Y 92.062,Z 810.07,A -85,B 0,C 180,E1 -27207.275,E2 -27207.275} C_VEL
LIN {X 0,Y 89.088,Z 810.381,A -85,B 0,C 180,E1 -27212.92,E2 -27212.92} C_VEL
LIN {X 0,Y 87.111,Z 810.903,A -85,B 0,C 180,E1 -27218.712,E2 -27218.712} C_VEL
LIN {X 0,Y 86.368,Z 810.717,A -85,B 0,C 180,E1 -27224.751,E2 -27224.751} C_VEL
LIN {X 0,Y 86.449,Z 810.707,A -85,B 0,C 180,E1 -27229.43,E2 -27229.43} C_VEL
LIN {X 0,Y 86.528,Z 810.705,A -85,B 0,C 180,E1 -27235.35,E2 -27235.35} C_VEL
LIN {X 0,Y 86.577,Z 810.701,A -85,B 0,C 180,E1 -27243.234,E2 -27243.234} C_VEL
LIN {X 0,Y 86.617,Z 810.695,A -85,B 0,C 180,E1 -27251.061,E2 -27251.061} C_VEL
LIN {X 0,Y 86.893,Z 810.652,A -85,B 0,C 180,E1 -27256.043,E2 -27256.043} C_VEL
LIN {X 0,Y 87.055,Z 810.641,A -85,B 0,C 180,E1 -27260.708,E2 -27260.708} C_VEL
LIN {X 0,Y 87.676,Z 810.565,A -85,B 0,C 180,E1 -27270,E2 -27270} C_VEL
LIN {X 0,Y 87.054,Z 810.641,A -85,B 0,C 180,E1 -27279.292,E2 -27279.292} C_VEL
LIN {X 0,Y 86.877,Z 810.654,A -85,B 0,C 180,E1 -27284.045,E2 -27284.045} C_VEL
LIN {X 0,Y 86.617,Z 810.695,A -85,B 0,C 180,E1 -27288.939,E2 -27288.939} C_VEL
LIN {X 0,Y 86.577,Z 810.701,A -85,B 0,C 180,E1 -27296.766,E2 -27296.766} C_VEL
LIN {X 0,Y 86.503,Z 810.71,A -85,B 0,C 180,E1 -27305.672,E2 -27305.672} C_VEL
LIN {X 0,Y 86.441,Z 810.714,A -85,B 0,C 180,E1 -27312.975,E2 -27312.975} C_VEL
LIN {X 0,Y 86.376,Z 810.717,A -85,B 0,C 180,E1 -27319.396,E2 -27319.396} C_VEL
LIN {X 0,Y 86.164,Z 810.752,A -85,B 0,C 180,E1 -27325.189,E2 -27325.189} C_VEL
LIN {X 0,Y 86.258,Z 810.734,A -85,B 0,C 180,E1 -27336.229,E2 -27336.229} C_VEL
LIN {X 0,Y 89.024,Z 823.773,A -85,B 0,C 180,E1 -27339.877,E2 -27339.877} C_VEL
LIN {X 0,Y 90.099,Z 828.665,A -85,B 0,C 180,E1 -27341.427,E2 -27341.427} C_VEL
LIN {X 0,Y 88.624,Z 840.18,A -85,B 0,C 180,E1 -27346.242,E2 -27346.242} C_VEL
LIN {X 0,Y 87.577,Z 851.044,A -85,B 0,C 180,E1 -27351.932,E2 -27351.932} C_VEL
LIN {X 0,Y 87.101,Z 861.779,A -85,B 0,C 180,E1 -27358.849,E2 -27358.849} C_VEL
LIN {X 0,Y 87.399,Z 870.608,A -85,B 0,C 180,E1 -27365.774,E2 -27365.774} C_VEL
LIN {X 0,Y 88.338,Z 877.883,A -85,B 0,C 180,E1 -27372.642,E2 -27372.642} C_VEL
LIN {X 0,Y 91.004,Z 885.575,A -85,B 0,C 180,E1 -27381.06,E2 -27381.06} C_VEL
LIN {X 0,Y 95.682,Z 891.936,A -85,B 0,C 180,E1 -27388.523,E2 -27388.523} C_VEL
LIN {X 0,Y 102.43,Z 897.633,A -85,B 0,C 180,E1 -27395.681,E2 -27395.681} C_VEL
LIN {X 0,Y 113.337,Z 903.327,A -85,B 0,C 180,E1 -27403.013,E2 -27403.013} C_VEL
LIN {X 0,Y 105.638,Z 901.309,A -85,B 0,C 180,E1 -27408.295,E2 -27408.295} C_VEL
LIN {X 0,Y 98.439,Z 898.224,A -85,B 0,C 180,E1 -27415.169,E2 -27415.169} C_VEL
LIN {X 0,Y 93.283,Z 894.239,A -85,B 0,C 180,E1 -27423.125,E2 -27423.125} C_VEL
LIN {X 0,Y 90.581,Z 889.298,A -85,B 0,C 180,E1 -27431.919,E2 -27431.919} C_VEL
LIN {X 0,Y 90.379,Z 883.148,A -85,B 0,C 180,E1 -27441.053,E2 -27441.053} C_VEL
LIN {X 0,Y 92.12,Z 876.215,A -85,B 0,C 180,E1 -27449.262,E2 -27449.262} C_VEL
LIN {X 0,Y 90.438,Z 883.05,A -85,B 0,C 180,E1 -27456.694,E2 -27456.694} C_VEL
LIN {X 0,Y 90.169,Z 889.454,A -85,B 0,C 180,E1 -27465.831,E2 -27465.831} C_VEL
LIN {X 0,Y 93.221,Z 895.623,A -85,B 0,C 180,E1 -27476.894,E2 -27476.894} C_VEL
LIN {X 0,Y 98.421,Z 899.498,A -85,B 0,C 180,E1 -27484.838,E2 -27484.838} C_VEL
LIN {X 0,Y 105.625,Z 902.519,A -85,B 0,C 180,E1 -27491.711,E2 -27491.711} C_VEL
LIN {X 0,Y 113.534,Z 904.51,A -85,B 0,C 180,E1 -27497.079,E2 -27497.079} C_VEL
LIN {X 0,Y 102.557,Z 898.872,A -85,B 0,C 180,E1 -27504.37,E2 -27504.37} C_VEL
LIN {X 0,Y 94.294,Z 891.615,A -85,B 0,C 180,E1 -27513.431,E2 -27513.431} C_VEL
LIN {X 0,Y 89.809,Z 884.434,A -85,B 0,C 180,E1 -27521.754,E2 -27521.754} C_VEL
LIN {X 0,Y 87.885,Z 877.096,A -85,B 0,C 180,E1 -27529.63,E2 -27529.63} C_VEL
LIN {X 0,Y 87.137,Z 869.42,A -85,B 0,C 180,E1 -27536.527,E2 -27536.527} C_VEL
LIN {X 0,Y 87.021,Z 860.233,A -85,B 0,C 180,E1 -27543.468,E2 -27543.468} C_VEL
LIN {X 0,Y 87.809,Z 848.922,A -85,B 0,C 180,E1 -27550.37,E2 -27550.37} C_VEL
LIN {X 0,Y 89.345,Z 836.226,A -85,B 0,C 180,E1 -27556.563,E2 -27556.563} C_VEL
LIN {X 0,Y 90.121,Z 830.328,A -85,B 0,C 180,E1 -27558.98,E2 -27558.98} C_VEL
LIN {X 0,Y 88.062,Z 820.042,A -85,B 0,C 180,E1 -27562.228,E2 -27562.228} C_VEL
LIN {X 0,Y 86.221,Z 810.744,A -85,B 0,C 180,E1 -27564.79,E2 -27564.79} C_VEL
LIN {X 0,Y 86.13,Z 810.756,A -85,B 0,C 180,E1 -27575.315,E2 -27575.315} C_VEL
LIN {X 0,Y 86.409,Z 810.719,A -85,B 0,C 180,E1 -27582.945,E2 -27582.945} C_VEL
LIN {X 0,Y 86.368,Z 810.717,A -85,B 0,C 180,E1 -27584.751,E2 -27584.751} C_VEL
LIN {X 0,Y 85.719,Z 810.802,A -85,B 0,C 180,E1 -27588.648,E2 -27588.648} C_VEL
LIN {X 0,Y 84.186,Z 810.997,A -85,B 0,C 180,E1 -27592.52,E2 -27592.52} C_VEL
LIN {X 0,Y 79.736,Z 811.553,A -85,B 0,C 180,E1 -27603.443,E2 -27603.443} C_VEL
LIN {X 0,Y 79.414,Z 811.579,A -85,B 0,C 180,E1 -27606.367,E2 -27606.367} C_VEL
LIN {X 0,Y 79.8,Z 811.536,A -85,B 0,C 180,E1 -27615.62,E2 -27615.62} C_VEL
LIN {X 0,Y 79.938,Z 811.527,A -85,B 0,C 180,E1 -27619.873,E2 -27619.873} C_VEL
LIN {X 0,Y 80.605,Z 811.445,A -85,B 0,C 180,E1 -27630,E2 -27630} C_VEL
LIN {X 0,Y 79.937,Z 811.527,A -85,B 0,C 180,E1 -27640.127,E2 -27640.127} C_VEL
LIN {X 0,Y 79.715,Z 811.55,A -85,B 0,C 180,E1 -27645.337,E2 -27645.337} C_VEL
LIN {X 0,Y 79.493,Z 811.578,A -85,B 0,C 180,E1 -27650.71,E2 -27650.71} C_VEL
LIN {X 0,Y 79.474,Z 811.585,A -85,B 0,C 180,E1 -27657.845,E2 -27657.845} C_VEL
LIN {X 0,Y 79.372,Z 811.589,A -85,B 0,C 180,E1 -27662.091,E2 -27662.091} C_VEL
LIN {X 0,Y 79.359,Z 811.596,A -85,B 0,C 180,E1 -27668.31,E2 -27668.31} C_VEL
LIN {X 0,Y 79.331,Z 811.604,A -85,B 0,C 180,E1 -27675.132,E2 -27675.132} C_VEL
LIN {X 0,Y 79.119,Z 811.629,A -85,B 0,C 180,E1 -27683.078,E2 -27683.078} C_VEL
LIN {X 0,Y 78.954,Z 811.641,A -85,B 0,C 180,E1 -27687.724,E2 -27687.724} C_VEL
LIN {X 0,Y 79.339,Z 811.592,A -85,B 0,C 180,E1 -27697.108,E2 -27697.108} C_VEL
LIN {X 0,Y 82.692,Z 826.601,A -85,B 0,C 180,E1 -27701.741,E2 -27701.741} C_VEL
LIN {X 0,Y 82.957,Z 829.304,A -85,B 0,C 180,E1 -27702.757,E2 -27702.757} C_VEL
LIN {X 0,Y 81.694,Z 839.672,A -85,B 0,C 180,E1 -27707.586,E2 -27707.586} C_VEL
LIN {X 0,Y 80.788,Z 850.599,A -85,B 0,C 180,E1 -27713.762,E2 -27713.762} C_VEL
LIN {X 0,Y 80.542,Z 859.665,A -85,B 0,C 180,E1 -27720.005,E2 -27720.005} C_VEL
LIN {X 0,Y 81.026,Z 868.69,A -85,B 0,C 180,E1 -27727.481,E2 -27727.481} C_VEL
LIN {X 0,Y 82.198,Z 876.138,A -85,B 0,C 180,E1 -27734.868,E2 -27734.868} C_VEL
LIN {X 0,Y 85.612,Z 884.44,A -85,B 0,C 180,E1 -27744.239,E2 -27744.239} C_VEL
LIN {X 0,Y 93.136,Z 892.975,A -85,B 0,C 180,E1 -27754.473,E2 -27754.473} C_VEL
LIN {X 0,Y 103.473,Z 899.722,A -85,B 0,C 180,E1 -27762.787,E2 -27762.787} C_VEL
LIN {X 0,Y 100.734,Z 898.99,A -85,B 0,C 180,E1 -27765.759,E2 -27765.759} C_VEL
LIN {X 0,Y 93.104,Z 895.606,A -85,B 0,C 180,E1 -27772.851,E2 -27772.851} C_VEL
LIN {X 0,Y 86.716,Z 890.347,A -85,B 0,C 180,E1 -27783.073,E2 -27783.073} C_VEL
LIN {X 0,Y 84.254,Z 884.646,A -85,B 0,C 180,E1 -27793.025,E2 -27793.025} C_VEL
LIN {X 0,Y 84.26,Z 879.708,A -85,B 0,C 180,E1 -27800.397,E2 -27800.397} C_VEL
LIN {X 0,Y 86.145,Z 872.429,A -85,B 0,C 180,E1 -27809.166,E2 -27809.166} C_VEL
LIN {X 0,Y 84.214,Z 880.344,A -85,B 0,C 180,E1 -27818.277,E2 -27818.277} C_VEL
LIN {X 0,Y 84.109,Z 886.238,A -85,B 0,C 180,E1 -27827.005,E2 -27827.005} C_VEL
LIN {X 0,Y 87.47,Z 892.765,A -85,B 0,C 180,E1 -27838.822,E2 -27838.822} C_VEL
LIN {X 0,Y 93.069,Z 896.925,A -85,B 0,C 180,E1 -27847.165,E2 -27847.165} C_VEL
LIN {X 0,Y 100.702,Z 900.219,A -85,B 0,C 180,E1 -27854.259,E2 -27854.259} C_VEL
LIN {X 0,Y 103.665,Z 900.992,A -85,B 0,C 180,E1 -27857.311,E2 -27857.311} C_VEL
LIN {X 0,Y 93.199,Z 894.268,A -85,B 0,C 180,E1 -27865.553,E2 -27865.553} C_VEL
LIN {X 0,Y 86.868,Z 887.648,A -85,B 0,C 180,E1 -27873.573,E2 -27873.573} C_VEL
LIN {X 0,Y 82.756,Z 879.798,A -85,B 0,C 180,E1 -27882.703,E2 -27882.703} C_VEL
LIN {X 0,Y 81.226,Z 872.886,A -85,B 0,C 180,E1 -27890.03,E2 -27890.03} C_VEL
LIN {X 0,Y 80.551,Z 866.037,A -85,B 0,C 180,E1 -27896.243,E2 -27896.243} C_VEL
LIN {X 0,Y 80.501,Z 856.235,A -85,B 0,C 180,E1 -27903.749,E2 -27903.749} C_VEL
LIN {X 0,Y 81.193,Z 845.396,A -85,B 0,C 180,E1 -27910.594,E2 -27910.594} C_VEL
LIN {X 0,Y 82.643,Z 833.166,A -85,B 0,C 180,E1 -27916.674,E2 -27916.674} C_VEL
LIN {X 0,Y 83.004,Z 828.771,A -85,B 0,C 180,E1 -27918.507,E2 -27918.507} C_VEL
LIN {X 0,Y 79.971,Z 815.391,A -85,B 0,C 180,E1 -27922.81,E2 -27922.81} C_VEL
LIN {X 0,Y 79.281,Z 811.605,A -85,B 0,C 180,E1 -27924.025,E2 -27924.025} C_VEL
LIN {X 0,Y 78.896,Z 811.648,A -85,B 0,C 180,E1 -27932.302,E2 -27932.302} C_VEL
LIN {X 0,Y 79.13,Z 811.624,A -85,B 0,C 180,E1 -27938.434,E2 -27938.434} C_VEL
LIN {X 0,Y 79.329,Z 811.604,A -85,B 0,C 180,E1 -27945.125,E2 -27945.125} C_VEL
LIN {X 0,Y 79.381,Z 811.596,A -85,B 0,C 180,E1 -27952.818,E2 -27952.818} C_VEL
LIN {X 0,Y 79.372,Z 811.589,A -85,B 0,C 180,E1 -27957.909,E2 -27957.909} C_VEL
LIN {X 0,Y 79.517,Z 811.579,A -85,B 0,C 180,E1 -27963.774,E2 -27963.774} C_VEL
LIN {X 0,Y 79.414,Z 811.579,A -85,B 0,C 180,E1 -27966.367,E2 -27966.367} C_VEL
LIN {X 0,Y 79.078,Z 811.629,A -85,B 0,C 180,E1 -27969.197,E2 -27969.197} C_VEL
LIN {X 0,Y 78.268,Z 811.736,A -85,B 0,C 180,E1 -27972.004,E2 -27972.004} C_VEL
LIN {X 0,Y 75.97,Z 812.014,A -85,B 0,C 180,E1 -27977.668,E2 -27977.668} C_VEL
LIN {X 0,Y 73.397,Z 812.335,A -85,B 0,C 180,E1 -27986.82,E2 -27986.82} C_VEL
LIN {X 0,Y 73.53,Z 812.326,A -85,B 0,C 180,E1 -27989.976,E2 -27989.976} C_VEL
LIN {X 0,Y 72.831,Z 812.41,A -85,B 0,C 180,E1 -28001.128,E2 -28001.128} C_VEL
LIN {X 0,Y 72.553,Z 812.447,A -85,B 0,C 180,E1 -28006.894,E2 -28006.894} C_VEL
LIN {X 0,Y 72.379,Z 812.46,A -85,B 0,C 180,E1 -28012.855,E2 -28012.855} C_VEL
LIN {X 0,Y 72.37,Z 812.467,A -85,B 0,C 180,E1 -28019.085,E2 -28019.085} C_VEL
LIN {X 0,Y 72.289,Z 812.48,A -85,B 0,C 180,E1 -28025.685,E2 -28025.685} C_VEL
LIN {X 0,Y 72.212,Z 812.487,A -85,B 0,C 180,E1 -28032.943,E2 -28032.943} C_VEL
LIN {X 0,Y 72.097,Z 812.499,A -85,B 0,C 180,E1 -28041.246,E2 -28041.246} C_VEL
LIN {X 0,Y 71.853,Z 812.533,A -85,B 0,C 180,E1 -28051.679,E2 -28051.679} C_VEL
LIN {X 0,Y 72.5,Z 812.441,A -85,B 0,C 180,E1 -28058.366,E2 -28058.366} C_VEL
LIN {X 0,Y 75.957,Z 827.204,A -85,B 0,C 180,E1 -28063.287,E2 -28063.287} C_VEL
LIN {X 0,Y 75.57,Z 832.865,A -85,B 0,C 180,E1 -28065.876,E2 -28065.876} C_VEL
LIN {X 0,Y 74.415,Z 844.816,A -85,B 0,C 180,E1 -28072.544,E2 -28072.544} C_VEL
LIN {X 0,Y 74.059,Z 855.54,A -85,B 0,C 180,E1 -28080.006,E2 -28080.006} C_VEL
LIN {X 0,Y 74.473,Z 863.732,A -85,B 0,C 180,E1 -28086.78,E2 -28086.78} C_VEL
LIN {X 0,Y 75.712,Z 871.801,A -85,B 0,C 180,E1 -28094.795,E2 -28094.795} C_VEL
LIN {X 0,Y 79.014,Z 880.714,A -85,B 0,C 180,E1 -28104.998,E2 -28104.998} C_VEL
LIN {X 0,Y 85.996,Z 889.247,A -85,B 0,C 180,E1 -28115.189,E2 -28115.189} C_VEL
LIN {X 0,Y 93.858,Z 895.257,A -85,B 0,C 180,E1 -28122.375,E2 -28122.375} C_VEL
LIN {X 0,Y 94.564,Z 895.872,A -85,B 0,C 180,E1 -28124.18,E2 -28124.18} C_VEL
LIN {X 0,Y 86.298,Z 891.733,A -85,B 0,C 180,E1 -28132.353,E2 -28132.353} C_VEL
LIN {X 0,Y 81.083,Z 887.22,A -85,B 0,C 180,E1 -28141.033,E2 -28141.033} C_VEL
LIN {X 0,Y 78.319,Z 881.236,A -85,B 0,C 180,E1 -28151.695,E2 -28151.695} C_VEL
LIN {X 0,Y 78.372,Z 875.345,A -85,B 0,C 180,E1 -28160.577,E2 -28160.577} C_VEL
LIN {X 0,Y 80.273,Z 868.456,A -85,B 0,C 180,E1 -28169.105,E2 -28169.105} C_VEL
LIN {X 0,Y 78.078,Z 877.768,A -85,B 0,C 180,E1 -28180.371,E2 -28180.371} C_VEL
LIN {X 0,Y 78.583,Z 884.322,A -85,B 0,C 180,E1 -28190.961,E2 -28190.961} C_VEL
LIN {X 0,Y 81.939,Z 889.678,A -85,B 0,C 180,E1 -28200.973,E2 -28200.973} C_VEL
LIN {X 0,Y 87.956,Z 894.12,A -85,B 0,C 180,E1 -28209.735,E2 -28209.735} C_VEL
LIN {X 0,Y 94.59,Z 897.181,A -85,B 0,C 180,E1 -28215.912,E2 -28215.912} C_VEL
LIN {X 0,Y 93.982,Z 896.598,A -85,B 0,C 180,E1 -28217.694,E2 -28217.694} C_VEL
LIN {X 0,Y 83.44,Z 888.106,A -85,B 0,C 180,E1 -28227.944,E2 -28227.944} C_VEL
LIN {X 0,Y 76.947,Z 877.983,A -85,B 0,C 180,E1 -28239.965,E2 -28239.965} C_VEL
LIN {X 0,Y 75.087,Z 870.861,A -85,B 0,C 180,E1 -28247.837,E2 -28247.837} C_VEL
LIN {X 0,Y 74.172,Z 863.909,A -85,B 0,C 180,E1 -28254.557,E2 -28254.557} C_VEL
LIN {X 0,Y 73.913,Z 855.664,A -85,B 0,C 180,E1 -28261.357,E2 -28261.357} C_VEL
LIN {X 0,Y 74.43,Z 844.726,A -85,B 0,C 180,E1 -28268.821,E2 -28268.821} C_VEL
LIN {X 0,Y 75.665,Z 832.682,A -85,B 0,C 180,E1 -28275.482,E2 -28275.482} C_VEL
LIN {X 0,Y 76.064,Z 828.823,A -85,B 0,C 180,E1 -28277.291,E2 -28277.291} C_VEL
LIN {X 0,Y 73.042,Z 815.899,A -85,B 0,C 180,E1 -28281.765,E2 -28281.765} C_VEL
LIN {X 0,Y 72.401,Z 812.455,A -85,B 0,C 180,E1 -28282.841,E2 -28282.841} C_VEL
LIN {X 0,Y 71.943,Z 812.523,A -85,B 0,C 180,E1 -28295.875,E2 -28295.875} C_VEL
LIN {X 0,Y 72.118,Z 812.498,A -85,B 0,C 180,E1 -28303.004,E2 -28303.004} C_VEL
LIN {X 0,Y 72.284,Z 812.474,A -85,B 0,C 180,E1 -28311.052,E2 -28311.052} C_VEL
LIN {X 0,Y 72.289,Z 812.48,A -85,B 0,C 180,E1 -28314.315,E2 -28314.315} C_VEL
LIN {X 0,Y 72.368,Z 812.467,A -85,B 0,C 180,E1 -28320.95,E2 -28320.95} C_VEL
LIN {X 0,Y 72.38,Z 812.46,A -85,B 0,C 180,E1 -28327.145,E2 -28327.145} C_VEL
LIN {X 0,Y 72.697,Z 812.422,A -85,B 0,C 180,E1 -28335.16,E2 -28335.16} C_VEL
LIN {X 0,Y 72.831,Z 812.41,A -85,B 0,C 180,E1 -28338.872,E2 -28338.872} C_VEL
LIN {X 0,Y 73.53,Z 812.326,A -85,B 0,C 180,E1 -28349.976,E2 -28349.976} C_VEL
LIN {X 0,Y 73.522,Z 812.351,A -85,B 0,C 180,E1 -28352.991,E2 -28352.991} C_VEL
LIN {X 0,Y 72.2,Z 812.54,A -85,B 0,C 180,E1 -28357.488,E2 -28357.488} C_VEL
LIN {X 0,Y 70.046,Z 812.816,A -85,B 0,C 180,E1 -28361.968,E2 -28361.968} C_VEL
LIN {X 0,Y 65.759,Z 813.316,A -85,B 0,C 180,E1 -28371.999,E2 -28371.999} C_VEL
LIN {X 0,Y 65.223,Z 813.358,A -85,B 0,C 180,E1 -28375.64,E2 -28375.64} C_VEL
LIN {X 0,Y 65.189,Z 813.356,A -85,B 0,C 180,E1 -28382.619,E2 -28382.619} C_VEL
LIN {X 0,Y 65.158,Z 813.359,A -85,B 0,C 180,E1 -28390.983,E2 -28390.983} C_VEL
LIN {X 0,Y 65.022,Z 813.376,A -85,B 0,C 180,E1 -28399.579,E2 -28399.579} C_VEL
LIN {X 0,Y 64.785,Z 813.408,A -85,B 0,C 180,E1 -28410.211,E2 -28410.211} C_VEL
LIN {X 0,Y 65.784,Z 813.45,A -85,B 0,C 180,E1 -28420.03,E2 -28420.03} C_VEL
LIN {X 0,Y 68.903,Z 826.297,A -85,B 0,C 180,E1 -28424.599,E2 -28424.599} C_VEL
LIN {X 0,Y 69.133,Z 827.938,A -85,B 0,C 180,E1 -28425.283,E2 -28425.283} C_VEL
LIN {X 0,Y 68.002,Z 840.644,A -85,B 0,C 180,E1 -28432.584,E2 -28432.584} C_VEL
LIN {X 0,Y 67.642,Z 851.091,A -85,B 0,C 180,E1 -28440.006,E2 -28440.006} C_VEL
LIN {X 0,Y 68.155,Z 859.755,A -85,B 0,C 180,E1 -28447.412,E2 -28447.412} C_VEL
LIN {X 0,Y 69.283,Z 867.049,A -85,B 0,C 180,E1 -28454.696,E2 -28454.696} C_VEL
LIN {X 0,Y 72.033,Z 875.492,A -85,B 0,C 180,E1 -28464.504,E2 -28464.504} C_VEL
LIN {X 0,Y 76.875,Z 882.799,A -85,B 0,C 180,E1 -28473.272,E2 -28473.272} C_VEL
LIN {X 0,Y 85.865,Z 890.944,A -85,B 0,C 180,E1 -28482.917,E2 -28482.917} C_VEL
LIN {X 0,Y 86.041,Z 891.263,A -85,B 0,C 180,E1 -28484.599,E2 -28484.599} C_VEL
LIN {X 0,Y 78.282,Z 886.399,A -85,B 0,C 180,E1 -28493.909,E2 -28493.909} C_VEL
LIN {X 0,Y 73.693,Z 880.756,A -85,B 0,C 180,E1 -28504.586,E2 -28504.586} C_VEL
LIN {X 0,Y 72.319,Z 873.787,A -85,B 0,C 180,E1 -28516.385,E2 -28516.385} C_VEL
LIN {X 0,Y 74.542,Z 864.254,A -85,B 0,C 180,E1 -28529.066,E2 -28529.066} C_VEL
LIN {X 0,Y 72.709,Z 869.683,A -85,B 0,C 180,E1 -28535.547,E2 -28535.547} C_VEL
LIN {X 0,Y 72.119,Z 875.044,A -85,B 0,C 180,E1 -28542.944,E2 -28542.944} C_VEL
LIN {X 0,Y 73.511,Z 882.297,A -85,B 0,C 180,E1 -28555.482,E2 -28555.482} C_VEL
LIN {X 0,Y 79.581,Z 888.908,A -85,B 0,C 180,E1 -28568.184,E2 -28568.184} C_VEL
LIN {X 0,Y 86.044,Z 892.639,A -85,B 0,C 180,E1 -28575.46,E2 -28575.46} C_VEL
LIN {X 0,Y 85.913,Z 892.357,A -85,B 0,C 180,E1 -28577.148,E2 -28577.148} C_VEL
LIN {X 0,Y 76.861,Z 884.279,A -85,B 0,C 180,E1 -28586.721,E2 -28586.721} C_VEL
LIN {X 0,Y 71.41,Z 875.922,A -85,B 0,C 180,E1 -28596.811,E2 -28596.811} C_VEL
LIN {X 0,Y 69.128,Z 868.771,A -85,B 0,C 180,E1 -28605.27,E2 -28605.27} C_VEL
LIN {X 0,Y 67.97,Z 861.518,A -85,B 0,C 180,E1 -28612.568,E2 -28612.568} C_VEL
LIN {X 0,Y 67.504,Z 853.057,A -85,B 0,C 180,E1 -28619.994,E2 -28619.994} C_VEL
LIN {X 0,Y 67.787,Z 842.897,A -85,B 0,C 180,E1 -28627.44,E2 -28627.44} C_VEL
LIN {X 0,Y 68.936,Z 830.461,A -85,B 0,C 180,E1 -28634.76,E2 -28634.76} C_VEL
LIN {X 0,Y 69.104,Z 829.053,A -85,B 0,C 180,E1 -28635.478,E2 -28635.478} C_VEL
LIN {X 0,Y 67.661,Z 822.351,A -85,B 0,C 180,E1 -28638.15,E2 -28638.15} C_VEL
LIN {X 0,Y 65.562,Z 813.307,A -85,B 0,C 180,E1 -28641.5,E2 -28641.5} C_VEL
LIN {X 0,Y 64.73,Z 813.414,A -85,B 0,C 180,E1 -28652.871,E2 -28652.871} C_VEL
LIN {X 0,Y 65.016,Z 813.377,A -85,B 0,C 180,E1 -28660.827,E2 -28660.827} C_VEL
LIN {X 0,Y 65.18,Z 813.356,A -85,B 0,C 180,E1 -28669.688,E2 -28669.688} C_VEL
LIN {X 0,Y 65.248,Z 813.348,A -85,B 0,C 180,E1 -28679.495,E2 -28679.495} C_VEL
LIN {X 0,Y 65.228,Z 813.358,A -85,B 0,C 180,E1 -28684.47,E2 -28684.47} C_VEL
LIN {X 0,Y 65.604,Z 813.307,A -85,B 0,C 180,E1 -28694.585,E2 -28694.585} C_VEL
LIN {X 0,Y 65.73,Z 813.289,A -85,B 0,C 180,E1 -28697.652,E2 -28697.652} C_VEL
LIN {X 0,Y 66.433,Z 813.211,A -85,B 0,C 180,E1 -28710,E2 -28710} C_VEL
LIN {X 0,Y 65.73,Z 813.289,A -85,B 0,C 180,E1 -28722.348,E2 -28722.348} C_VEL
LIN {X 0,Y 65.363,Z 813.343,A -85,B 0,C 180,E1 -28728.818,E2 -28728.818} C_VEL
LIN {X 0,Y 65.223,Z 813.358,A -85,B 0,C 180,E1 -28735.64,E2 -28735.64} C_VEL
LIN {X 0,Y 64.778,Z 813.413,A -85,B 0,C 180,E1 -28739.086,E2 -28739.086} C_VEL
LIN {X 0,Y 63.314,Z 813.596,A -85,B 0,C 180,E1 -28744.23,E2 -28744.23} C_VEL
LIN {X 0,Y 60.041,Z 814.003,A -85,B 0,C 180,E1 -28753.1,E2 -28753.1} C_VEL
LIN {X 0,Y 57.656,Z 814.288,A -85,B 0,C 180,E1 -28764.907,E2 -28764.907} C_VEL
LIN {X 0,Y 57.753,Z 814.286,A -85,B 0,C 180,E1 -28770.881,E2 -28770.881} C_VEL
LIN {X 0,Y 59.092,Z 814.133,A -85,B 0,C 180,E1 -28782.077,E2 -28782.077} C_VEL
LIN {X 0,Y 62.316,Z 826.761,A -85,B 0,C 180,E1 -28786.971,E2 -28786.971} C_VEL
LIN {X 0,Y 61.493,Z 838.591,A -85,B 0,C 180,E1 -28794.267,E2 -28794.267} C_VEL
LIN {X 0,Y 61.46,Z 850.059,A -85,B 0,C 180,E1 -28803.284,E2 -28803.284} C_VEL
LIN {X 0,Y 62.39,Z 858.77,A -85,B 0,C 180,E1 -28811.376,E2 -28811.376} C_VEL
LIN {X 0,Y 63.934,Z 865.974,A -85,B 0,C 180,E1 -28819.262,E2 -28819.262} C_VEL
LIN {X 0,Y 68.283,Z 875.538,A -85,B 0,C 180,E1 -28830.979,E2 -28830.979} C_VEL
LIN {X 0,Y 76.025,Z 884.284,A -85,B 0,C 180,E1 -28841.429,E2 -28841.429} C_VEL
LIN {X 0,Y 77.843,Z 885.827,A -85,B 0,C 180,E1 -28843.183,E2 -28843.183} C_VEL
LIN {X 0,Y 78.65,Z 886.501,A -85,B 0,C 180,E1 -28844.368,E2 -28844.368} C_VEL
LIN {X 0,Y 71.656,Z 881.423,A -85,B 0,C 180,E1 -28853.951,E2 -28853.951} C_VEL
LIN {X 0,Y 67.55,Z 875.405,A -85,B 0,C 180,E1 -28865.407,E2 -28865.407} C_VEL
LIN {X 0,Y 66.688,Z 868.052,A -85,B 0,C 180,E1 -28877.832,E2 -28877.832} C_VEL
LIN {X 0,Y 68.912,Z 859.951,A -85,B 0,C 180,E1 -28889.087,E2 -28889.087} C_VEL
LIN {X 0,Y 66.904,Z 865.435,A -85,B 0,C 180,E1 -28896.03,E2 -28896.03} C_VEL
LIN {X 0,Y 66.39,Z 871.995,A -85,B 0,C 180,E1 -28905.665,E2 -28905.665} C_VEL
LIN {X 0,Y 68.115,Z 878.607,A -85,B 0,C 180,E1 -28917.665,E2 -28917.665} C_VEL
LIN {X 0,Y 72.947,Z 884.185,A -85,B 0,C 180,E1 -28928.546,E2 -28928.546} C_VEL
LIN {X 0,Y 78.576,Z 887.911,A -85,B 0,C 180,E1 -28935.687,E2 -28935.687} C_VEL
LIN {X 0,Y 77.914,Z 887.347,A -85,B 0,C 180,E1 -28936.738,E2 -28936.738} C_VEL
LIN {X 0,Y 68.954,Z 878.199,A -85,B 0,C 180,E1 -28947.643,E2 -28947.643} C_VEL
LIN {X 0,Y 64.202,Z 868.939,A -85,B 0,C 180,E1 -28959.153,E2 -28959.153} C_VEL
LIN {X 0,Y 62.188,Z 860.66,A -85,B 0,C 180,E1 -28968.587,E2 -28968.587} C_VEL
LIN {X 0,Y 61.281,Z 852.104,A -85,B 0,C 180,E1 -28976.706,E2 -28976.706} C_VEL
LIN {X 0,Y 61.283,Z 840.831,A -85,B 0,C 180,E1 -28985.752,E2 -28985.752} C_VEL
LIN {X 0,Y 62.135,Z 829.582,A -85,B 0,C 180,E1 -28993.068,E2 -28993.068} C_VEL
LIN {X 0,Y 62.078,Z 827.182,A -85,B 0,C 180,E1 -28994.332,E2 -28994.332} C_VEL
LIN {X 0,Y 58.83,Z 814.154,A -85,B 0,C 180,E1 -28999.6,E2 -28999.6} C_VEL
LIN {X 0,Y 57.695,Z 814.288,A -85,B 0,C 180,E1 -29011.493,E2 -29011.493} C_VEL
LIN {X 0,Y 57.738,Z 814.291,A -85,B 0,C 180,E1 -29017.48,E2 -29017.48} C_VEL
LIN {X 0,Y 57.953,Z 814.263,A -85,B 0,C 180,E1 -29026.677,E2 -29026.677} C_VEL
LIN {X 0,Y 58.016,Z 814.257,A -85,B 0,C 180,E1 -29032.721,E2 -29032.721} C_VEL
LIN {X 0,Y 58.151,Z 814.232,A -85,B 0,C 180,E1 -29037.765,E2 -29037.765} C_VEL
LIN {X 0,Y 58.143,Z 814.239,A -85,B 0,C 180,E1 -29041.086,E2 -29041.086} C_VEL
LIN {X 0,Y 58.498,Z 814.195,A -85,B 0,C 180,E1 -29053.944,E2 -29053.944} C_VEL
LIN {X 0,Y 58.769,Z 814.16,A -85,B 0,C 180,E1 -29063.132,E2 -29063.132} C_VEL
LIN {X 0,Y 59.327,Z 814.096,A -85,B 0,C 180,E1 -29070,E2 -29070} C_VEL
LIN {X 0,Y 58.768,Z 814.16,A -85,B 0,C 180,E1 -29076.868,E2 -29076.868} C_VEL
LIN {X 0,Y 58.498,Z 814.195,A -85,B 0,C 180,E1 -29086.056,E2 -29086.056} C_VEL
LIN {X 0,Y 58.143,Z 814.239,A -85,B 0,C 180,E1 -29098.914,E2 -29098.914} C_VEL
LIN {X 0,Y 58.151,Z 814.232,A -85,B 0,C 180,E1 -29102.235,E2 -29102.235} C_VEL
LIN {X 0,Y 58.017,Z 814.257,A -85,B 0,C 180,E1 -29107.279,E2 -29107.279} C_VEL
LIN {X 0,Y 57.9,Z 814.27,A -85,B 0,C 180,E1 -29116.744,E2 -29116.744} C_VEL
LIN {X 0,Y 57.656,Z 814.288,A -85,B 0,C 180,E1 -29124.907,E2 -29124.907} C_VEL
LIN {X 0,Y 56.925,Z 814.386,A -85,B 0,C 180,E1 -29127.268,E2 -29127.268} C_VEL
LIN {X 0,Y 54.171,Z 814.731,A -85,B 0,C 180,E1 -29130.707,E2 -29130.707} C_VEL
LIN {X 0,Y 51.353,Z 815.084,A -85,B 0,C 180,E1 -29134.941,E2 -29134.941} C_VEL
LIN {X 0,Y 51.051,Z 815.113,A -85,B 0,C 180,E1 -29137.273,E2 -29137.273} C_VEL
LIN {X 0,Y 52.579,Z 815.113,A -85,B 0,C 180,E1 -29144.833,E2 -29144.833} C_VEL
LIN {X 0,Y 55.367,Z 825.257,A -85,B 0,C 180,E1 -29149.031,E2 -29149.031} C_VEL
LIN {X 0,Y 55.622,Z 827.105,A -85,B 0,C 180,E1 -29150.002,E2 -29150.002} C_VEL
LIN {X 0,Y 55.086,Z 839.611,A -85,B 0,C 180,E1 -29159.094,E2 -29159.094} C_VEL
LIN {X 0,Y 55.767,Z 850.831,A -85,B 0,C 180,E1 -29169.071,E2 -29169.071} C_VEL
LIN {X 0,Y 57.363,Z 859.081,A -85,B 0,C 180,E1 -29177.843,E2 -29177.843} C_VEL
LIN {X 0,Y 60.177,Z 867.263,A -85,B 0,C 180,E1 -29187.857,E2 -29187.857} C_VEL
LIN {X 0,Y 68.498,Z 878.597,A -85,B 0,C 180,E1 -29201.836,E2 -29201.836} C_VEL
LIN {X 0,Y 70.639,Z 880.562,A -85,B 0,C 180,E1 -29204.15,E2 -29204.15} C_VEL
LIN {X 0,Y 70.356,Z 880.464,A -85,B 0,C 180,E1 -29205.633,E2 -29205.633} C_VEL
LIN {X 0,Y 64.133,Z 874.648,A -85,B 0,C 180,E1 -29216.775,E2 -29216.775} C_VEL
LIN {X 0,Y 61.285,Z 867.775,A -85,B 0,C 180,E1 -29229.877,E2 -29229.877} C_VEL
LIN {X 0,Y 61.591,Z 860.37,A -85,B 0,C 180,E1 -29241.8,E2 -29241.8} C_VEL
LIN {X 0,Y 63.493,Z 855.367,A -85,B 0,C 180,E1 -29248.95,E2 -29248.95} C_VEL
LIN {X 0,Y 61.278,Z 860.916,A -85,B 0,C 180,E1 -29256.586,E2 -29256.586} C_VEL
LIN {X 0,Y 60.847,Z 868.096,A -85,B 0,C 180,E1 -29267.495,E2 -29267.495} C_VEL
LIN {X 0,Y 63.906,Z 876.31,A -85,B 0,C 180,E1 -29283.359,E2 -29283.359} C_VEL
LIN {X 0,Y 70.261,Z 881.988,A -85,B 0,C 180,E1 -29294.442,E2 -29294.442} C_VEL
LIN {X 0,Y 70.61,Z 882.153,A -85,B 0,C 180,E1 -29295.827,E2 -29295.827} C_VEL
LIN {X 0,Y 62.075,Z 872.49,A -85,B 0,C 180,E1 -29307.459,E2 -29307.459} C_VEL
LIN {X 0,Y 58.003,Z 863.777,A -85,B 0,C 180,E1 -29318.677,E2 -29318.677} C_VEL
LIN {X 0,Y 56.087,Z 856.217,A -85,B 0,C 180,E1 -29327.326,E2 -29327.326} C_VEL
LIN {X 0,Y 55.003,Z 847.194,A -85,B 0,C 180,E1 -29336.33,E2 -29336.33} C_VEL
LIN {X 0,Y 54.925,Z 837.353,A -85,B 0,C 180,E1 -29344.579,E2 -29344.579} C_VEL
LIN {X 0,Y 55.465,Z 828.353,A -85,B 0,C 180,E1 -29350.949,E2 -29350.949} C_VEL
LIN {X 0,Y 55.049,Z 825.499,A -85,B 0,C 180,E1 -29352.434,E2 -29352.434} C_VEL
LIN {X 0,Y 52.256,Z 814.975,A -85,B 0,C 180,E1 -29356.915,E2 -29356.915} C_VEL
LIN {X 0,Y 50.605,Z 815.175,A -85,B 0,C 180,E1 -29373.736,E2 -29373.736} C_VEL
LIN {X 0,Y 50.849,Z 815.149,A -85,B 0,C 180,E1 -29383.703,E2 -29383.703} C_VEL
LIN {X 0,Y 50.908,Z 815.142,A -85,B 0,C 180,E1 -29386.348,E2 -29386.348} C_VEL
LIN {X 0,Y 51.04,Z 815.12,A -85,B 0,C 180,E1 -29396.579,E2 -29396.579} C_VEL
LIN {X 0,Y 51.013,Z 815.124,A -85,B 0,C 180,E1 -29405.587,E2 -29405.587} C_VEL
LIN {X 0,Y 51.451,Z 815.07,A -85,B 0,C 180,E1 -29414.146,E2 -29414.146} C_VEL
LIN {X 0,Y 51.649,Z 815.05,A -85,B 0,C 180,E1 -29422.179,E2 -29422.179} C_VEL
LIN {X 0,Y 52.214,Z 814.982,A -85,B 0,C 180,E1 -29430,E2 -29430} C_VEL
LIN {X 0,Y 51.648,Z 815.05,A -85,B 0,C 180,E1 -29437.821,E2 -29437.821} C_VEL
LIN {X 0,Y 51.355,Z 815.086,A -85,B 0,C 180,E1 -29446.703,E2 -29446.703} C_VEL
LIN {X 0,Y 51.013,Z 815.124,A -85,B 0,C 180,E1 -29454.413,E2 -29454.413} C_VEL
LIN {X 0,Y 50.995,Z 815.129,A -85,B 0,C 180,E1 -29464.233,E2 -29464.233} C_VEL
LIN {X 0,Y 50.909,Z 815.141,A -85,B 0,C 180,E1 -29473.65,E2 -29473.65} C_VEL
LIN {X 0,Y 50.851,Z 815.149,A -85,B 0,C 180,E1 -29476.299,E2 -29476.299} C_VEL
LIN {X 0,Y 50.628,Z 815.172,A -85,B 0,C 180,E1 -29486.398,E2 -29486.398} C_VEL
LIN {X 0,Y 51.051,Z 815.113,A -85,B 0,C 180,E1 -29497.273,E2 -29497.273} C_VEL
LIN {X 0,Y 51.114,Z 815.687,A -85,B 0,C 180,E1 -29500.814,E2 -29500.814} C_VEL
LIN {X 0,Y 50.603,Z 817.695,A -85,B 0,C 180,E1 -29504.94,E2 -29504.94} C_VEL
LIN {X 0,Y 49.57,Z 821.73,A -85,B 0,C 180,E1 -29509.78,E2 -29509.78} C_VEL
LIN {X 0,Y 48.506,Z 830.57,A -85,B 0,C 180,E1 -29516.927,E2 -29516.927} C_VEL
LIN {X 0,Y 49.028,Z 837.889,A -85,B 0,C 180,E1 -29522.693,E2 -29522.693} C_VEL
LIN {X 0,Y 50.404,Z 849.462,A -85,B 0,C 180,E1 -29534.131,E2 -29534.131} C_VEL
LIN {X 0,Y 52.563,Z 857.731,A -85,B 0,C 180,E1 -29543.656,E2 -29543.656} C_VEL
LIN {X 0,Y 57.12,Z 867.015,A -85,B 0,C 180,E1 -29555.772,E2 -29555.772} C_VEL
LIN {X 0,Y 63.154,Z 874.261,A -85,B 0,C 180,E1 -29564.656,E2 -29564.656} C_VEL
LIN {X 0,Y 62.433,Z 873.746,A -85,B 0,C 180,E1 -29567.513,E2 -29567.513} C_VEL
LIN {X 0,Y 57.247,Z 867.177,A -85,B 0,C 180,E1 -29580.589,E2 -29580.589} C_VEL
LIN {X 0,Y 55.745,Z 860.848,A -85,B 0,C 180,E1 -29592.581,E2 -29592.581} C_VEL
LIN {X 0,Y 57.237,Z 852.275,A -85,B 0,C 180,E1 -29606.128,E2 -29606.128} C_VEL
LIN {X 0,Y 58.259,Z 850.574,A -85,B 0,C 180,E1 -29608.886,E2 -29608.886} C_VEL
LIN {X 0,Y 55.813,Z 856.225,A -85,B 0,C 180,E1 -29617.234,E2 -29617.234} C_VEL
LIN {X 0,Y 55.418,Z 862.434,A -85,B 0,C 180,E1 -29626.969,E2 -29626.969} C_VEL
LIN {X 0,Y 57.837,Z 870.504,A -85,B 0,C 180,E1 -29642.734,E2 -29642.734} C_VEL
LIN {X 0,Y 62.244,Z 875.338,A -85,B 0,C 180,E1 -29652.646,E2 -29652.646} C_VEL
LIN {X 0,Y 62.953,Z 875.837,A -85,B 0,C 180,E1 -29655.401,E2 -29655.401} C_VEL
LIN {X 0,Y 55.439,Z 866.284,A -85,B 0,C 180,E1 -29667.391,E2 -29667.391} C_VEL
LIN {X 0,Y 52.353,Z 859.613,A -85,B 0,C 180,E1 -29676.243,E2 -29676.243} C_VEL
LIN {X 0,Y 50.166,Z 851.487,A -85,B 0,C 180,E1 -29685.8,E2 -29685.8} C_VEL
LIN {X 0,Y 48.805,Z 840.642,A -85,B 0,C 180,E1 -29696.896,E2 -29696.896} C_VEL
LIN {X 0,Y 48.799,Z 829.734,A -85,B 0,C 180,E1 -29706.192,E2 -29706.192} C_VEL
LIN {X 0,Y 48.932,Z 826.963,A -85,B 0,C 180,E1 -29708.249,E2 -29708.249} C_VEL
LIN {X 0,Y 45.803,Z 815.771,A -85,B 0,C 180,E1 -29713.58,E2 -29713.58} C_VEL
LIN {X 0,Y 43.489,Z 816.068,A -85,B 0,C 180,E1 -29736.096,E2 -29736.096} C_VEL
LIN {X 0,Y 43.549,Z 816.049,A -85,B 0,C 180,E1 -29740.193,E2 -29740.193} C_VEL
LIN {X 0,Y 43.75,Z 816.024,A -85,B 0,C 180,E1 -29750.017,E2 -29750.017} C_VEL
LIN {X 0,Y 43.804,Z 816.028,A -85,B 0,C 180,E1 -29753.326,E2 -29753.326} C_VEL
LIN {X 0,Y 43.832,Z 816.02,A -85,B 0,C 180,E1 -29761.248,E2 -29761.248} C_VEL
LIN {X 0,Y 44.21,Z 815.978,A -85,B 0,C 180,E1 -29772.485,E2 -29772.485} C_VEL
LIN {X 0,Y 44.508,Z 815.941,A -85,B 0,C 180,E1 -29780.915,E2 -29780.915} C_VEL
LIN {X 0,Y 45.091,Z 815.869,A -85,B 0,C 180,E1 -29790,E2 -29790} C_VEL
LIN {X 0,Y 44.507,Z 815.941,A -85,B 0,C 180,E1 -29799.085,E2 -29799.085} C_VEL
LIN {X 0,Y 44.134,Z 815.987,A -85,B 0,C 180,E1 -29808.571,E2 -29808.571} C_VEL
LIN {X 0,Y 43.833,Z 816.02,A -85,B 0,C 180,E1 -29818.752,E2 -29818.752} C_VEL
LIN {X 0,Y 43.804,Z 816.028,A -85,B 0,C 180,E1 -29826.675,E2 -29826.675} C_VEL
LIN {X 0,Y 43.751,Z 816.024,A -85,B 0,C 180,E1 -29829.982,E2 -29829.982} C_VEL
LIN {X 0,Y 43.556,Z 816.049,A -85,B 0,C 180,E1 -29839.816,E2 -29839.816} C_VEL
LIN {X 0,Y 43.576,Z 816.051,A -85,B 0,C 180,E1 -29851.074,E2 -29851.074} C_VEL
LIN {X 0,Y 46.193,Z 815.726,A -85,B 0,C 180,E1 -29868.351,E2 -29868.351} C_VEL
LIN {X 0,Y 49.117,Z 825.532,A -85,B 0,C 180,E1 -29872.816,E2 -29872.816} C_VEL
LIN {X 0,Y 49.028,Z 837.889,A -85,B 0,C 180,E1 -29882.693,E2 -29882.693} C_VEL
LIN {X 0,Y 48.789,Z 842.278,A -85,B 0,C 180,E1 -29887.306,E2 -29887.306} C_VEL
LIN {X 0,Y 48.155,Z 846.075,A -85,B 0,C 180,E1 -29892.663,E2 -29892.663} C_VEL
LIN {X 0,Y 48.173,Z 855.012,A -85,B 0,C 180,E1 -29908.629,E2 -29908.629} C_VEL
LIN {X 0,Y 49.147,Z 857.41,A -85,B 0,C 180,E1 -29912.262,E2 -29912.262} C_VEL
LIN {X 0,Y 55.324,Z 866.612,A -85,B 0,C 180,E1 -29924.332,E2 -29924.332} C_VEL
LIN {X 0,Y 56.01,Z 867.404,A -85,B 0,C 180,E1 -29925.276,E2 -29925.276} C_VEL
LIN {X 0,Y 55.675,Z 867.136,A -85,B 0,C 180,E1 -29928.497,E2 -29928.497} C_VEL
LIN {X 0,Y 51.375,Z 860.237,A -85,B 0,C 180,E1 -29942.761,E2 -29942.761} C_VEL
LIN {X 0,Y 50.627,Z 852.959,A -85,B 0,C 180,E1 -29956.379,E2 -29956.379} C_VEL
LIN {X 0,Y 52.151,Z 847.269,A -85,B 0,C 180,E1 -29965.749,E2 -29965.749} C_VEL
LIN {X 0,Y 53.253,Z 845.568,A -85,B 0,C 180,E1 -29968.782,E2 -29968.782} C_VEL
LIN {X 0,Y 50.815,Z 850.194,A -85,B 0,C 180,E1 -29976.202,E2 -29976.202} C_VEL
LIN {X 0,Y 50.328,Z 858.625,A -85,B 0,C 180,E1 -29990.433,E2 -29990.433} C_VEL
LIN {X 0,Y 52.157,Z 864.589,A -85,B 0,C 180,E1 -30002.615,E2 -30002.615} C_VEL
LIN {X 0,Y 56.028,Z 869.375,A -85,B 0,C 180,E1 -30012.815,E2 -30012.815} C_VEL
LIN {X 0,Y 55.187,Z 868.414,A -85,B 0,C 180,E1 -30015.529,E2 -30015.529} C_VEL
LIN {X 0,Y 48.285,Z 858.014,A -85,B 0,C 180,E1 -30029.364,E2 -30029.364} C_VEL
LIN {X 0,Y 45.798,Z 851.79,A -85,B 0,C 180,E1 -30037.426,E2 -30037.426} C_VEL
LIN {X 0,Y 43.548,Z 842.308,A -85,B 0,C 180,E1 -30048.352,E2 -30048.352} C_VEL
LIN {X 0,Y 42.638,Z 832.028,A -85,B 0,C 180,E1 -30058.81,E2 -30058.81} C_VEL
LIN {X 0,Y 42.589,Z 826.758,A -85,B 0,C 180,E1 -30063.546,E2 -30063.546} C_VEL
LIN {X 0,Y 41.936,Z 823.902,A -85,B 0,C 180,E1 -30065.327,E2 -30065.327} C_VEL
LIN {X 0,Y 39.649,Z 816.547,A -85,B 0,C 180,E1 -30068.966,E2 -30068.966} C_VEL
LIN {X 0,Y 36.484,Z 816.93,A -85,B 0,C 180,E1 -30099.598,E2 -30099.598} C_VEL
LIN {X 0,Y 36.673,Z 816.906,A -85,B 0,C 180,E1 -30110.029,E2 -30110.029} C_VEL
LIN {X 0,Y 36.694,Z 816.912,A -85,B 0,C 180,E1 -30114.928,E2 -30114.928} C_VEL
LIN {X 0,Y 37.042,Z 816.871,A -85,B 0,C 180,E1 -30131.523,E2 -30131.523} C_VEL
LIN {X 0,Y 37.307,Z 816.831,A -85,B 0,C 180,E1 -30139.142,E2 -30139.142} C_VEL
LIN {X 0,Y 37.954,Z 816.758,A -85,B 0,C 180,E1 -30150,E2 -30150} C_VEL
LIN {X 0,Y 37.307,Z 816.831,A -85,B 0,C 180,E1 -30160.859,E2 -30160.859} C_VEL
LIN {X 0,Y 37.042,Z 816.871,A -85,B 0,C 180,E1 -30168.477,E2 -30168.477} C_VEL
LIN {X 0,Y 36.694,Z 816.912,A -85,B 0,C 180,E1 -30185.071,E2 -30185.071} C_VEL
LIN {X 0,Y 36.673,Z 816.906,A -85,B 0,C 180,E1 -30189.973,E2 -30189.973} C_VEL
LIN {X 0,Y 36.494,Z 816.928,A -85,B 0,C 180,E1 -30200.384,E2 -30200.384} C_VEL
LIN {X 0,Y 37.214,Z 816.845,A -85,B 0,C 180,E1 -30220.78,E2 -30220.78} C_VEL
LIN {X 0,Y 40.163,Z 816.476,A -85,B 0,C 180,E1 -30233.227,E2 -30233.227} C_VEL
LIN {X 0,Y 42.878,Z 825.132,A -85,B 0,C 180,E1 -30237.429,E2 -30237.429} C_VEL
LIN {X 0,Y 43.429,Z 836.707,A -85,B 0,C 180,E1 -30248.15,E2 -30248.15} C_VEL
LIN {X 0,Y 45.52,Z 847.969,A -85,B 0,C 180,E1 -30260.337,E2 -30260.337} C_VEL
LIN {X 0,Y 48.394,Z 855.795,A -85,B 0,C 180,E1 -30270.077,E2 -30270.077} C_VEL
LIN {X 0,Y 49.147,Z 857.41,A -85,B 0,C 180,E1 -30272.262,E2 -30272.262} C_VEL
LIN {X 0,Y 49.68,Z 859.015,A -85,B 0,C 180,E1 -30275.598,E2 -30275.598} C_VEL
LIN {X 0,Y 49.618,Z 859.788,A -85,B 0,C 180,E1 -30279.444,E2 -30279.444} C_VEL
LIN {X 0,Y 49.205,Z 859.845,A -85,B 0,C 180,E1 -30284.278,E2 -30284.278} C_VEL
LIN {X 0,Y 48.254,Z 858.729,A -85,B 0,C 180,E1 -30291.142,E2 -30291.142} C_VEL
LIN {X 0,Y 47.076,Z 856.469,A -85,B 0,C 180,E1 -30297.674,E2 -30297.674} C_VEL
LIN {X 0,Y 45.562,Z 849.391,A -85,B 0,C 180,E1 -30312.031,E2 -30312.031} C_VEL
LIN {X 0,Y 47.079,Z 842.394,A -85,B 0,C 180,E1 -30324.724,E2 -30324.724} C_VEL
LIN {X 0,Y 48.388,Z 840.407,A -85,B 0,C 180,E1 -30328.718,E2 -30328.718} C_VEL
LIN {X 0,Y 45.733,Z 845.042,A -85,B 0,C 180,E1 -30336.894,E2 -30336.894} C_VEL
LIN {X 0,Y 45.507,Z 854.547,A -85,B 0,C 180,E1 -30354.286,E2 -30354.286} C_VEL
LIN {X 0,Y 49.212,Z 862.025,A -85,B 0,C 180,E1 -30370.723,E2 -30370.723} C_VEL
LIN {X 0,Y 49.552,Z 862.43,A -85,B 0,C 180,E1 -30373.031,E2 -30373.031} C_VEL
LIN {X 0,Y 44.183,Z 854.819,A -85,B 0,C 180,E1 -30383.369,E2 -30383.369} C_VEL
LIN {X 0,Y 41.081,Z 848.249,A -85,B 0,C 180,E1 -30392.025,E2 -30392.025} C_VEL
LIN {X 0,Y 38.243,Z 839.132,A -85,B 0,C 180,E1 -30403.302,E2 -30403.302} C_VEL
LIN {X 0,Y 36.795,Z 828.65,A -85,B 0,C 180,E1 -30414.852,E2 -30414.852} C_VEL
LIN {X 0,Y 36.663,Z 825.611,A -85,B 0,C 180,E1 -30417.929,E2 -30417.929} C_VEL
LIN {X 0,Y 35.516,Z 822.048,A -85,B 0,C 180,E1 -30419.988,E2 -30419.988} C_VEL
LIN {X 0,Y 33.828,Z 817.259,A -85,B 0,C 180,E1 -30422.703,E2 -30422.703} C_VEL
LIN {X 0,Y 29.404,Z 817.681,A -85,B 0,C 180,E1 -30448.541,E2 -30448.541} C_VEL
LIN {X 0,Y 29.386,Z 817.685,A -85,B 0,C 180,E1 -30465.828,E2 -30465.828} C_VEL
LIN {X 0,Y 29.475,Z 817.675,A -85,B 0,C 180,E1 -30481.518,E2 -30481.518} C_VEL
LIN {X 0,Y 29.851,Z 817.64,A -85,B 0,C 180,E1 -30490.305,E2 -30490.305} C_VEL
LIN {X 0,Y 30.089,Z 817.614,A -85,B 0,C 180,E1 -30496.492,E2 -30496.492} C_VEL
LIN {X 0,Y 30.776,Z 817.554,A -85,B 0,C 180,E1 -30510,E2 -30510} C_VEL
LIN {X 0,Y 30.089,Z 817.614,A -85,B 0,C 180,E1 -30523.508,E2 -30523.508} C_VEL
LIN {X 0,Y 29.851,Z 817.64,A -85,B 0,C 180,E1 -30529.695,E2 -30529.695} C_VEL
LIN {X 0,Y 29.475,Z 817.675,A -85,B 0,C 180,E1 -30538.482,E2 -30538.482} C_VEL
LIN {X 0,Y 29.365,Z 817.685,A -85,B 0,C 180,E1 -30555.89,E2 -30555.89} C_VEL
LIN {X 0,Y 29.371,Z 817.684,A -85,B 0,C 180,E1 -30571.424,E2 -30571.424} C_VEL
LIN {X 0,Y 33.956,Z 817.248,A -85,B 0,C 180,E1 -30598.53,E2 -30598.53} C_VEL
LIN {X 0,Y 34.668,Z 817.261,A -85,B 0,C 180,E1 -30600.012,E2 -30600.012} C_VEL
LIN {X 0,Y 37.032,Z 823.944,A -85,B 0,C 180,E1 -30603.25,E2 -30603.25} C_VEL
LIN {X 0,Y 38.237,Z 835.028,A -85,B 0,C 180,E1 -30614.65,E2 -30614.65} C_VEL
LIN {X 0,Y 41.179,Z 845.656,A -85,B 0,C 180,E1 -30627.183,E2 -30627.183} C_VEL
LIN {X 0,Y 44.439,Z 852.832,A -85,B 0,C 180,E1 -30636.386,E2 -30636.386} C_VEL
LIN {X 0,Y 49.87,Z 860.72,A -85,B 0,C 180,E1 -30646.972,E2 -30646.972} C_VEL
LIN {X 0,Y 49.33,Z 860.084,A -85,B 0,C 180,E1 -30649.958,E2 -30649.958} C_VEL
LIN {X 0,Y 47.076,Z 856.469,A -85,B 0,C 180,E1 -30657.674,E2 -30657.674} C_VEL
LIN {X 0,Y 45.898,Z 854.125,A -85,B 0,C 180,E1 -30661.342,E2 -30661.342} C_VEL
LIN {X 0,Y 43.35,Z 849.148,A -85,B 0,C 180,E1 -30666.173,E2 -30666.173} C_VEL
LIN {X 0,Y 41.216,Z 843.961,A -85,B 0,C 180,E1 -30671.37,E2 -30671.37} C_VEL
LIN {X 0,Y 40.927,Z 841.29,A -85,B 0,C 180,E1 -30675.518,E2 -30675.518} C_VEL
LIN {X 0,Y 42.39,Z 836.964,A -85,B 0,C 180,E1 -30684.231,E2 -30684.231} C_VEL
LIN {X 0,Y 43.75,Z 835.024,A -85,B 0,C 180,E1 -30688.563,E2 -30688.563} C_VEL
LIN {X 0,Y 41.062,Z 839.346,A -85,B 0,C 180,E1 -30697.128,E2 -30697.128} C_VEL
LIN {X 0,Y 40.433,Z 847.843,A -85,B 0,C 180,E1 -30713.851,E2 -30713.851} C_VEL
LIN {X 0,Y 42.878,Z 854.136,A -85,B 0,C 180,E1 -30727.924,E2 -30727.924} C_VEL
LIN {X 0,Y 43.543,Z 855.154,A -85,B 0,C 180,E1 -30730.212,E2 -30730.212} C_VEL
LIN {X 0,Y 42.857,Z 854.306,A -85,B 0,C 180,E1 -30732.423,E2 -30732.423} C_VEL
LIN {X 0,Y 38.796,Z 848.223,A -85,B 0,C 180,E1 -30740.638,E2 -30740.638} C_VEL
LIN {X 0,Y 34.57,Z 838.817,A -85,B 0,C 180,E1 -30752.708,E2 -30752.708} C_VEL
LIN {X 0,Y 31.838,Z 828.345,A -85,B 0,C 180,E1 -30765.608,E2 -30765.608} C_VEL
LIN {X 0,Y 31.247,Z 824.429,A -85,B 0,C 180,E1 -30770.235,E2 -30770.235} C_VEL
LIN {X 0,Y 28.589,Z 817.757,A -85,B 0,C 180,E1 -30773.892,E2 -30773.892} C_VEL
LIN {X 0,Y 22.671,Z 818.07,A -85,B 0,C 180,E1 -30801.563,E2 -30801.563} C_VEL
LIN {X 0,Y 22.051,Z 818.089,A -85,B 0,C 180,E1 -30819.575,E2 -30819.575} C_VEL
LIN {X 0,Y 22.087,Z 818.088,A -85,B 0,C 180,E1 -30830.477,E2 -30830.477} C_VEL
LIN {X 0,Y 22.795,Z 818.066,A -85,B 0,C 180,E1 -30852.042,E2 -30852.042} C_VEL
LIN {X 0,Y 23.552,Z 818.042,A -85,B 0,C 180,E1 -30870,E2 -30870} C_VEL
LIN {X 0,Y 22.795,Z 818.066,A -85,B 0,C 180,E1 -30887.958,E2 -30887.958} C_VEL
LIN {X 0,Y 22.09,Z 818.088,A -85,B 0,C 180,E1 -30909.517,E2 -30909.517} C_VEL
LIN {X 0,Y 22.045,Z 818.089,A -85,B 0,C 180,E1 -30920.412,E2 -30920.412} C_VEL
LIN {X 0,Y 22.909,Z 818.062,A -85,B 0,C 180,E1 -30942.154,E2 -30942.154} C_VEL
LIN {X 0,Y 28.287,Z 817.785,A -85,B 0,C 180,E1 -30966.374,E2 -30966.374} C_VEL
LIN {X 0,Y 29.76,Z 817.823,A -85,B 0,C 180,E1 -30969.117,E2 -30969.117} C_VEL
LIN {X 0,Y 31.773,Z 822.913,A -85,B 0,C 180,E1 -30971.367,E2 -30971.367} C_VEL
LIN {X 0,Y 33.819,Z 832.963,A -85,B 0,C 180,E1 -30982.945,E2 -30982.945} C_VEL
LIN {X 0,Y 37.265,Z 842.447,A -85,B 0,C 180,E1 -30994.47,E2 -30994.47} C_VEL
LIN {X 0,Y 41.023,Z 849.309,A -85,B 0,C 180,E1 -31003.27,E2 -31003.27} C_VEL
LIN {X 0,Y 43.066,Z 852.245,A -85,B 0,C 180,E1 -31007.273,E2 -31007.273} C_VEL
LIN {X 0,Y 43.848,Z 853.22,A -85,B 0,C 180,E1 -31010.124,E2 -31010.124} C_VEL
LIN {X 0,Y 41.14,Z 846.849,A -85,B 0,C 180,E1 -31024.326,E2 -31024.326} C_VEL
LIN {X 0,Y 40.927,Z 841.29,A -85,B 0,C 180,E1 -31035.518,E2 -31035.518} C_VEL
LIN {X 0,Y 40.719,Z 839.555,A -85,B 0,C 180,E1 -31040.064,E2 -31040.064} C_VEL
LIN {X 0,Y 39.888,Z 838.54,A -85,B 0,C 180,E1 -31045.027,E2 -31045.027} C_VEL
LIN {X 0,Y 38.219,Z 838.142,A -85,B 0,C 180,E1 -31053.117,E2 -31053.117} C_VEL
LIN {X 0,Y 36.658,Z 838.959,A -85,B 0,C 180,E1 -31062.023,E2 -31062.023} C_VEL
LIN {X 0,Y 35.869,Z 840.797,A -85,B 0,C 180,E1 -31071.324,E2 -31071.324} C_VEL
LIN {X 0,Y 36.32,Z 843.716,A -85,B 0,C 180,E1 -31079.957,E2 -31079.957} C_VEL
LIN {X 0,Y 37.514,Z 846.597,A -85,B 0,C 180,E1 -31086.487,E2 -31086.487} C_VEL
LIN {X 0,Y 37.637,Z 847.006,A -85,B 0,C 180,E1 -31089.265,E2 -31089.265} C_VEL
LIN {X 0,Y 32.47,Z 838.821,A -85,B 0,C 180,E1 -31099.493,E2 -31099.493} C_VEL
LIN {X 0,Y 28.353,Z 828.702,A -85,B 0,C 180,E1 -31112.289,E2 -31112.289} C_VEL
LIN {X 0,Y 26.695,Z 822.902,A -85,B 0,C 180,E1 -31119.163,E2 -31119.163} C_VEL
LIN {X 0,Y 24.587,Z 818.011,A -85,B 0,C 180,E1 -31121.224,E2 -31121.224} C_VEL
LIN {X 0,Y 15.042,Z 818.178,A -85,B 0,C 180,E1 -31167.823,E2 -31167.823} C_VEL
LIN {X 0,Y 15.015,Z 818.178,A -85,B 0,C 180,E1 -31202.092,E2 -31202.092} C_VEL
LIN {X 0,Y 15.233,Z 818.178,A -85,B 0,C 180,E1 -31207.255,E2 -31207.255} C_VEL
LIN {X 0,Y 16.227,Z 818.178,A -85,B 0,C 180,E1 -31230,E2 -31230} C_VEL
LIN {X 0,Y 15.234,Z 818.178,A -85,B 0,C 180,E1 -31252.748,E2 -31252.748} C_VEL
LIN {X 0,Y 15.016,Z 818.178,A -85,B 0,C 180,E1 -31257.906,E2 -31257.906} C_VEL
LIN {X 0,Y 15.012,Z 818.178,A -85,B 0,C 180,E1 -31292.117,E2 -31292.117} C_VEL
LIN {X 0,Y 23.271,Z 818.051,A -85,B 0,C 180,E1 -31337.596,E2 -31337.596} C_VEL
LIN {X 0,Y 25.948,Z 818.067,A -85,B 0,C 180,E1 -31341.478,E2 -31341.478} C_VEL
LIN {X 0,Y 27.428,Z 821.58,A -85,B 0,C 180,E1 -31342.62,E2 -31342.62} C_VEL
LIN {X 0,Y 29.078,Z 827.191,A -85,B 0,C 180,E1 -31348.923,E2 -31348.923} C_VEL
LIN {X 0,Y 32.763,Z 836.363,A -85,B 0,C 180,E1 -31360.071,E2 -31360.071} C_VEL
LIN {X 0,Y 37.217,Z 843.864,A -85,B 0,C 180,E1 -31369.073,E2 -31369.073} C_VEL
LIN {X 0,Y 38.143,Z 845.034,A -85,B 0,C 180,E1 -31372.742,E2 -31372.742} C_VEL
LIN {X 0,Y 36.283,Z 836.761,A -85,B 0,C 180,E1 -31391.306,E2 -31391.306} C_VEL
LIN {X 0,Y 37.909,Z 831.394,A -85,B 0,C 180,E1 -31403.546,E2 -31403.546} C_VEL
LIN {X 0,Y 39.415,Z 829.438,A -85,B 0,C 180,E1 -31408.34,E2 -31408.34} C_VEL
LIN {X 0,Y 37.013,Z 832.555,A -85,B 0,C 180,E1 -31415.448,E2 -31415.448} C_VEL
LIN {X 0,Y 35.464,Z 839.281,A -85,B 0,C 180,E1 -31430.289,E2 -31430.289} C_VEL
LIN {X 0,Y 36.32,Z 843.716,A -85,B 0,C 180,E1 -31439.957,E2 -31439.957} C_VEL
LIN {X 0,Y 35.753,Z 843.012,A -85,B 0,C 180,E1 -31440.621,E2 -31440.621} C_VEL
LIN {X 0,Y 33.794,Z 839.429,A -85,B 0,C 180,E1 -31438.338,E2 -31438.338} C_VEL
LIN {X 0,Y 31.633,Z 831.877,A -85,B 0,C 180,E1 -31427.256,E2 -31427.256} C_VEL
LIN {X 0,Y 31.94,Z 828.577,A -85,B 0,C 180,E1 -31420.64,E2 -31420.64} C_VEL
LIN {X 0,Y 32.377,Z 827.414,A -85,B 0,C 180,E1 -31417.896,E2 -31417.896} C_VEL
LIN {X 0,Y 35.33,Z 823.634,A -85,B 0,C 180,E1 -31408.036,E2 -31408.036} C_VEL
LIN {X 0,Y 32.74,Z 827.508,A -85,B 0,C 180,E1 -31397.604,E2 -31397.604} C_VEL
LIN {X 0,Y 32.304,Z 834.304,A -85,B 0,C 180,E1 -31380.511,E2 -31380.511} C_VEL
LIN {X 0,Y 32.617,Z 836.053,A -85,B 0,C 180,E1 -31373.924,E2 -31373.924} C_VEL
LIN {X 0,Y 27.024,Z 825.988,A -85,B 0,C 180,E1 -31363.073,E2 -31363.073} C_VEL
LIN {X 0,Y 25.376,Z 822.151,A -85,B 0,C 180,E1 -31358.567,E2 -31358.567} C_VEL
LIN {X 0,Y 24.701,Z 820.49,A -85,B 0,C 180,E1 -31357.221,E2 -31357.221} C_VEL
LIN {X 0,Y 23.422,Z 818.046,A -85,B 0,C 180,E1 -31356.9,E2 -31356.9} C_VEL
LIN {X 0,Y 15.468,Z 818.178,A -85,B 0,C 180,E1 -31347.054,E2 -31347.054} C_VEL
LIN {X 0,Y 7.738,Z 818.178,A -85,B 0,C 180,E1 -31295.262,E2 -31295.262} C_VEL
LIN {X 0,Y 7.737,Z 818.178,A -85,B 0,C 180,E1 -31254.843,E2 -31254.843} C_VEL
LIN {X 0,Y 8.658,Z 818.178,A -85,B 0,C 180,E1 -31230,E2 -31230} C_VEL
LIN {X 0,Y 7.738,Z 818.178,A -85,B 0,C 180,E1 -31205.128,E2 -31205.128} C_VEL
LIN {X 0,Y 7.749,Z 818.178,A -85,B 0,C 180,E1 -31164.908,E2 -31164.908} C_VEL
LIN {X 0,Y 15.743,Z 818.178,A -85,B 0,C 180,E1 -31113.232,E2 -31113.232} C_VEL
LIN {X 0,Y 22.123,Z 818.236,A -85,B 0,C 180,E1 -31104.822,E2 -31104.822} C_VEL
LIN {X 0,Y 23.966,Z 822.391,A -85,B 0,C 180,E1 -31104.07,E2 -31104.07} C_VEL
LIN {X 0,Y 28.529,Z 832.281,A -85,B 0,C 180,E1 -31092.329,E2 -31092.329} C_VEL
LIN {X 0,Y 32.311,Z 838.366,A -85,B 0,C 180,E1 -31085.536,E2 -31085.536} C_VEL
LIN {X 0,Y 31.257,Z 830.758,A -85,B 0,C 180,E1 -31066.327,E2 -31066.327} C_VEL
LIN {X 0,Y 32.377,Z 827.414,A -85,B 0,C 180,E1 -31057.896,E2 -31057.896} C_VEL
LIN {X 0,Y 32.531,Z 825.634,A -85,B 0,C 180,E1 -31053.727,E2 -31053.727} C_VEL
LIN {X 0,Y 31.485,Z 823.384,A -85,B 0,C 180,E1 -31047.982,E2 -31047.982} C_VEL
LIN {X 0,Y 29.778,Z 821.828,A -85,B 0,C 180,E1 -31040.831,E2 -31040.831} C_VEL
LIN {X 0,Y 28.725,Z 821.934,A -85,B 0,C 180,E1 -31035.176,E2 -31035.176} C_VEL
LIN {X 0,Y 28.462,Z 822.418,A -85,B 0,C 180,E1 -31033.109,E2 -31033.109} C_VEL
LIN {X 0,Y 28.084,Z 824.337,A -85,B 0,C 180,E1 -31027.405,E2 -31027.405} C_VEL
LIN {X 0,Y 27.889,Z 826.322,A -85,B 0,C 180,E1 -31019.735,E2 -31019.735} C_VEL
LIN {X 0,Y 24.729,Z 820.645,A -85,B 0,C 180,E1 -31014.621,E2 -31014.621} C_VEL
LIN {X 0,Y 23.318,Z 818.049,A -85,B 0,C 180,E1 -31014.347,E2 -31014.347} C_VEL
